Yaskawa INFORM job: A_ROOF_SIDE_0617_2_PAINT_59.JBI

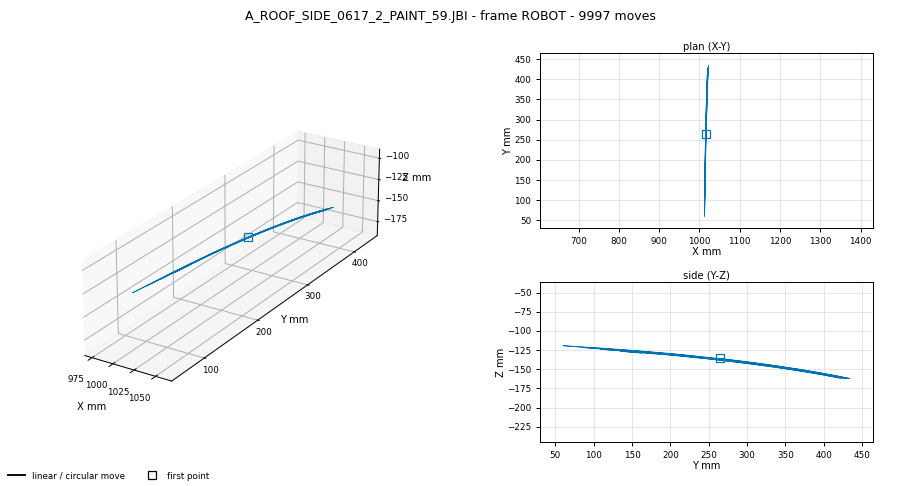
[picture p0: tool path of A_ROOF_SIDE_0617_2_PAINT_59.JBI in frame ROBOT, 9997 of 9997 moves have a stored position in this frame; points joined in program order, loops and branches not executed]
/JOB
//NAME A_ROOF_SIDE_0617_2_PAINT59
//POS
///NPOS 9997,0,0,0,0,0
///TOOL 1
///USER 0
///POSTYPE ROBOT
///RECTAN
///RCONF 1,0,0,0,0,0,0,0,0,0,0,0,0,0,0,0,0,0,0,0,0,0,0,0
C00000=1016.839,264.302,-135.724,169.198,51.675,159.894
C00001=1016.844,264.534,-135.751,169.203,51.669,159.893
C00002=1016.850,264.783,-135.779,169.208,51.663,159.893
C00003=1016.856,265.032,-135.809,169.212,51.657,159.892
C00004=1016.862,265.280,-135.837,169.217,51.651,159.892
C00005=1016.868,265.528,-135.866,169.222,51.644,159.891
C00006=1016.874,265.776,-135.895,169.228,51.638,159.891
C00007=1016.880,266.025,-135.923,169.233,51.632,159.891
C00008=1016.885,266.273,-135.953,169.237,51.626,159.890
C00009=1016.891,266.520,-135.982,169.242,51.620,159.890
C00010=1016.897,266.769,-136.010,169.247,51.614,159.889
C00011=1016.903,267.017,-136.039,169.252,51.607,159.889
C00012=1016.909,267.265,-136.068,169.257,51.602,159.888
C00013=1016.914,267.515,-136.097,169.262,51.596,159.888
C00014=1016.921,267.763,-136.126,169.267,51.589,159.887
C00015=1016.926,268.010,-136.155,169.272,51.583,159.887
C00016=1016.933,268.258,-136.184,169.277,51.577,159.887
C00017=1016.938,268.507,-136.213,169.282,51.571,159.886
C00018=1016.944,268.755,-136.242,169.287,51.565,159.886
C00019=1016.950,269.004,-136.271,169.292,51.559,159.885
C00020=1016.957,269.252,-136.300,169.297,51.553,159.885
C00021=1016.962,269.499,-136.329,169.302,51.547,159.884
C00022=1016.968,269.748,-136.358,169.306,51.541,159.884
C00023=1016.974,269.996,-136.387,169.311,51.535,159.883
C00024=1016.980,270.244,-136.417,169.317,51.529,159.883
C00025=1016.986,270.492,-136.446,169.322,51.523,159.883
C00026=1016.991,270.741,-136.476,169.327,51.517,159.882
C00027=1016.998,270.989,-136.505,169.332,51.511,159.882
C00028=1017.004,271.237,-136.534,169.337,51.505,159.882
C00029=1017.009,271.485,-136.563,169.342,51.500,159.881
C00030=1017.016,271.734,-136.592,169.347,51.494,159.881
C00031=1017.021,271.982,-136.622,169.352,51.488,159.880
C00032=1017.027,272.230,-136.651,169.357,51.482,159.880
C00033=1017.033,272.478,-136.680,169.362,51.476,159.880
C00034=1017.038,272.726,-136.709,169.367,51.470,159.879
C00035=1017.045,272.974,-136.738,169.372,51.464,159.879
C00036=1017.050,273.223,-136.768,169.377,51.459,159.879
C00037=1017.056,273.471,-136.797,169.382,51.453,159.878
C00038=1017.062,273.719,-136.827,169.387,51.447,159.878
C00039=1017.069,273.967,-136.856,169.392,51.441,159.877
C00040=1017.074,274.215,-136.886,169.398,51.435,159.877
C00041=1017.080,274.463,-136.915,169.403,51.429,159.877
C00042=1017.086,274.712,-136.945,169.408,51.423,159.876
C00043=1017.093,274.961,-136.974,169.414,51.418,159.876
C00044=1017.098,275.208,-137.005,169.419,51.412,159.876
C00045=1017.105,275.456,-137.034,169.424,51.407,159.875
C00046=1017.110,275.705,-137.063,169.429,51.401,159.875
C00047=1017.117,275.952,-137.093,169.434,51.395,159.875
C00048=1017.122,276.201,-137.123,169.439,51.389,159.874
C00049=1017.129,276.449,-137.152,169.444,51.384,159.874
C00050=1017.134,276.697,-137.182,169.449,51.378,159.874
C00051=1017.140,276.945,-137.212,169.454,51.372,159.873
C00052=1017.146,277.193,-137.241,169.459,51.367,159.873
C00053=1017.152,277.441,-137.271,169.464,51.361,159.873
C00054=1017.158,277.676,-137.300,169.469,51.357,159.872
C00055=1017.163,277.911,-137.328,169.474,51.351,159.872
C00056=1017.168,278.147,-137.356,169.479,51.346,159.872
C00057=1017.175,278.382,-137.385,169.484,51.341,159.871
C00058=1017.180,278.617,-137.413,169.489,51.335,159.871
C00059=1017.186,278.852,-137.442,169.494,51.330,159.871
C00060=1017.191,279.088,-137.470,169.498,51.325,159.871
C00061=1017.197,279.322,-137.498,169.503,51.319,159.870
C00062=1017.203,279.571,-137.528,169.509,51.314,159.870
C00063=1017.209,279.819,-137.558,169.514,51.308,159.870
C00064=1017.215,280.067,-137.588,169.519,51.303,159.869
C00065=1017.221,280.315,-137.618,169.524,51.297,159.869
C00066=1017.227,280.563,-137.648,169.530,51.292,159.869
C00067=1017.233,280.811,-137.678,169.535,51.286,159.868
C00068=1017.239,281.060,-137.708,169.540,51.281,159.868
C00069=1017.245,281.307,-137.738,169.546,51.276,159.868
C00070=1017.252,281.555,-137.768,169.551,51.270,159.868
C00071=1017.257,281.803,-137.798,169.556,51.265,159.868
C00072=1017.264,282.052,-137.829,169.561,51.259,159.867
C00073=1017.269,282.300,-137.859,169.566,51.254,159.867
C00074=1017.276,282.547,-137.889,169.572,51.249,159.867
C00075=1017.282,282.796,-137.919,169.577,51.243,159.866
C00076=1017.288,283.044,-137.949,169.582,51.238,159.866
C00077=1017.294,283.292,-137.979,169.588,51.233,159.866
C00078=1017.300,283.540,-138.009,169.593,51.227,159.866
C00079=1017.307,283.788,-138.040,169.598,51.222,159.865
C00080=1017.312,284.036,-138.070,169.604,51.217,159.865
C00081=1017.319,284.285,-138.100,169.609,51.211,159.865
C00082=1017.325,284.533,-138.130,169.614,51.206,159.865
C00083=1017.331,284.780,-138.160,169.619,51.201,159.864
C00084=1017.337,285.028,-138.191,169.625,51.196,159.864
C00085=1017.343,285.277,-138.221,169.629,51.191,159.864
C00086=1017.349,285.525,-138.252,169.634,51.185,159.864
C00087=1017.355,285.773,-138.282,169.640,51.180,159.863
C00088=1017.362,286.020,-138.313,169.645,51.175,159.863
C00089=1017.367,286.268,-138.344,169.651,51.170,159.863
C00090=1017.374,286.517,-138.375,169.656,51.165,159.863
C00091=1017.380,286.764,-138.405,169.661,51.160,159.863
C00092=1017.386,287.013,-138.436,169.667,51.155,159.862
C00093=1017.392,287.261,-138.466,169.672,51.149,159.862
C00094=1017.398,287.509,-138.496,169.678,51.144,159.862
C00095=1017.404,287.757,-138.527,169.683,51.139,159.862
C00096=1017.410,288.004,-138.558,169.689,51.134,159.862
C00097=1017.417,288.253,-138.589,169.694,51.129,159.861
C00098=1017.422,288.501,-138.619,169.699,51.124,159.861
C00099=1017.429,288.749,-138.650,169.705,51.119,159.861
C00100=1017.434,288.997,-138.682,169.710,51.114,159.861
C00101=1017.441,289.245,-138.712,169.716,51.108,159.861
C00102=1017.446,289.493,-138.743,169.721,51.103,159.861
C00103=1017.453,289.741,-138.774,169.726,51.099,159.860
C00104=1017.459,289.989,-138.804,169.731,51.094,159.860
C00105=1017.465,290.237,-138.835,169.737,51.089,159.860
C00106=1017.472,290.485,-138.866,169.742,51.084,159.860
C00107=1017.478,290.733,-138.897,169.748,51.079,159.860
C00108=1017.484,290.980,-138.928,169.753,51.074,159.860
C00109=1017.490,291.229,-138.959,169.759,51.069,159.859
C00110=1017.496,291.477,-138.989,169.764,51.064,159.859
C00111=1017.502,291.725,-139.021,169.770,51.059,159.859
C00112=1017.508,291.972,-139.052,169.775,51.054,159.859
C00113=1017.515,292.221,-139.083,169.781,51.049,159.859
C00114=1017.520,292.462,-139.113,169.786,51.045,159.859
C00115=1017.527,292.703,-139.143,169.791,51.040,159.858
C00116=1017.533,292.944,-139.173,169.797,51.035,159.859
C00117=1017.539,293.186,-139.204,169.802,51.030,159.858
C00118=1017.545,293.427,-139.235,169.807,51.026,159.858
C00119=1017.551,293.668,-139.265,169.812,51.021,159.858
C00120=1017.556,293.910,-139.295,169.818,51.017,159.858
C00121=1017.563,294.151,-139.327,169.823,51.012,159.858
C00122=1017.568,294.398,-139.358,169.829,51.007,159.858
C00123=1017.574,294.647,-139.390,169.834,51.003,159.858
C00124=1017.580,294.894,-139.421,169.840,50.998,159.858
C00125=1017.586,295.143,-139.453,169.846,50.993,159.858
C00126=1017.593,295.390,-139.484,169.851,50.988,159.857
C00127=1017.598,295.638,-139.516,169.856,50.984,159.857
C00128=1017.605,295.886,-139.547,169.861,50.979,159.857
C00129=1017.611,296.134,-139.579,169.867,50.975,159.857
C00130=1017.617,296.381,-139.610,169.873,50.970,159.857
C00131=1017.623,296.629,-139.642,169.879,50.965,159.857
C00132=1017.630,296.877,-139.674,169.884,50.961,159.857
C00133=1017.635,297.125,-139.705,169.890,50.956,159.857
C00134=1017.641,297.373,-139.737,169.896,50.951,159.857
C00135=1017.648,297.621,-139.769,169.900,50.947,159.857
C00136=1017.654,297.869,-139.801,169.906,50.943,159.857
C00137=1017.660,298.116,-139.832,169.912,50.938,159.857
C00138=1017.666,298.365,-139.864,169.918,50.933,159.857
C00139=1017.673,298.613,-139.895,169.923,50.929,159.857
C00140=1017.679,298.861,-139.927,169.929,50.924,159.857
C00141=1017.685,299.109,-139.959,169.935,50.920,159.857
C00142=1017.691,299.356,-139.991,169.941,50.915,159.856
C00143=1017.697,299.604,-140.022,169.945,50.911,159.856
C00144=1017.703,299.852,-140.054,169.951,50.906,159.856
C00145=1017.710,300.100,-140.087,169.957,50.902,159.856
C00146=1017.716,300.348,-140.118,169.963,50.898,159.856
C00147=1017.722,300.596,-140.150,169.969,50.893,159.856
C00148=1017.729,300.843,-140.181,169.974,50.888,159.856
C00149=1017.734,301.091,-140.213,169.980,50.884,159.856
C00150=1017.742,301.339,-140.245,169.986,50.879,159.856
C00151=1017.748,301.587,-140.278,169.992,50.875,159.856
C00152=1017.754,301.835,-140.309,169.997,50.871,159.856
C00153=1017.761,302.082,-140.342,170.002,50.866,159.856
C00154=1017.767,302.331,-140.374,170.008,50.862,159.856
C00155=1017.773,302.579,-140.405,170.014,50.857,159.856
C00156=1017.780,302.826,-140.438,170.020,50.853,159.856
C00157=1017.786,303.074,-140.469,170.026,50.849,159.856
C00158=1017.792,303.322,-140.501,170.032,50.844,159.856
C00159=1017.799,303.570,-140.533,170.037,50.840,159.856
C00160=1017.805,303.818,-140.566,170.043,50.835,159.856
C00161=1017.812,304.065,-140.598,170.049,50.831,159.856
C00162=1017.818,304.313,-140.630,170.055,50.827,159.856
C00163=1017.825,304.561,-140.662,170.060,50.822,159.856
C00164=1017.831,304.809,-140.694,170.066,50.818,159.856
C00165=1017.837,305.057,-140.726,170.072,50.814,159.856
C00166=1017.844,305.304,-140.758,170.078,50.810,159.856
C00167=1017.851,305.552,-140.791,170.084,50.805,159.856
C00168=1017.857,305.800,-140.823,170.089,50.801,159.856
C00169=1017.864,306.047,-140.855,170.095,50.797,159.856
C00170=1017.870,306.296,-140.887,170.101,50.792,159.856
C00171=1017.877,306.543,-140.919,170.107,50.789,159.857
C00172=1017.883,306.791,-140.951,170.113,50.784,159.857
C00173=1017.890,307.038,-140.983,170.119,50.780,159.857
C00174=1017.896,307.291,-141.017,170.125,50.775,159.857
C00175=1017.903,307.544,-141.049,170.131,50.771,159.857
C00176=1017.910,307.796,-141.083,170.137,50.767,159.857
C00177=1017.917,308.049,-141.116,170.143,50.763,159.857
C00178=1017.923,308.297,-141.147,170.149,50.758,159.857
C00179=1017.930,308.544,-141.180,170.155,50.754,159.857
C00180=1017.937,308.792,-141.212,170.161,50.750,159.857
C00181=1017.943,309.039,-141.245,170.167,50.746,159.857
C00182=1017.950,309.287,-141.278,170.172,50.741,159.857
C00183=1017.957,309.535,-141.309,170.179,50.738,159.857
C00184=1017.963,309.783,-141.342,170.185,50.733,159.857
C00185=1017.969,310.031,-141.375,170.190,50.730,159.857
C00186=1017.976,310.278,-141.408,170.196,50.726,159.858
C00187=1017.981,310.525,-141.442,170.202,50.722,159.858
C00188=1017.988,310.774,-141.475,170.208,50.718,159.858
C00189=1017.994,311.021,-141.508,170.214,50.714,159.858
C00190=1018.001,311.269,-141.540,170.220,50.710,159.858
C00191=1018.007,311.517,-141.573,170.225,50.706,159.858
C00192=1018.013,311.764,-141.607,170.232,50.703,159.858
C00193=1018.020,312.012,-141.640,170.238,50.698,159.858
C00194=1018.026,312.260,-141.673,170.244,50.695,159.859
C00195=1018.033,312.507,-141.706,170.250,50.691,159.859
C00196=1018.039,312.754,-141.739,170.256,50.687,159.859
C00197=1018.045,313.003,-141.773,170.262,50.683,159.859
C00198=1018.051,313.250,-141.806,170.267,50.679,159.859
C00199=1018.058,313.497,-141.839,170.274,50.676,159.859
C00200=1018.065,313.746,-141.872,170.280,50.672,159.859
C00201=1018.072,313.993,-141.906,170.286,50.668,159.860
C00202=1018.077,314.241,-141.939,170.292,50.664,159.860
C00203=1018.084,314.489,-141.972,170.298,50.660,159.860
C00204=1018.091,314.736,-142.006,170.304,50.656,159.860
C00205=1018.097,314.983,-142.038,170.311,50.652,159.860
C00206=1018.103,315.231,-142.073,170.316,50.649,159.860
C00207=1018.110,315.479,-142.105,170.322,50.645,159.861
C00208=1018.117,315.727,-142.139,170.328,50.642,159.861
C00209=1018.123,315.974,-142.172,170.335,50.638,159.861
C00210=1018.130,316.221,-142.205,170.341,50.634,159.861
C00211=1018.136,316.470,-142.239,170.347,50.630,159.861
C00212=1018.143,316.717,-142.273,170.353,50.627,159.862
C00213=1018.149,316.965,-142.306,170.360,50.623,159.862
C00214=1018.156,317.212,-142.339,170.366,50.619,159.862
C00215=1018.162,317.460,-142.374,170.372,50.615,159.862
C00216=1018.169,317.708,-142.406,170.377,50.612,159.862
C00217=1018.176,317.955,-142.440,170.384,50.608,159.863
C00218=1018.183,318.202,-142.474,170.390,50.605,159.863
C00219=1018.189,318.451,-142.507,170.396,50.601,159.863
C00220=1018.196,318.699,-142.541,170.403,50.598,159.863
C00221=1018.203,318.946,-142.575,170.409,50.594,159.864
C00222=1018.209,319.194,-142.608,170.415,50.590,159.864
C00223=1018.216,319.441,-142.641,170.421,50.587,159.864
C00224=1018.222,319.689,-142.676,170.428,50.583,159.864
C00225=1018.230,319.937,-142.709,170.434,50.579,159.864
C00226=1018.236,320.184,-142.742,170.441,50.576,159.865
C00227=1018.243,320.432,-142.776,170.447,50.572,159.865
C00228=1018.249,320.679,-142.810,170.453,50.569,159.865
C00229=1018.256,320.927,-142.844,170.459,50.565,159.865
C00230=1018.263,321.174,-142.878,170.466,50.562,159.866
C00231=1018.271,321.422,-142.912,170.472,50.558,159.866
C00232=1018.276,321.669,-142.946,170.478,50.554,159.866
C00233=1018.284,321.917,-142.979,170.484,50.552,159.867
C00234=1018.291,322.175,-143.014,170.491,50.548,159.867
C00235=1018.298,322.433,-143.049,170.498,50.544,159.867
C00236=1018.305,322.691,-143.084,170.504,50.540,159.867
C00237=1018.312,322.949,-143.120,170.511,50.537,159.868
C00238=1018.319,323.197,-143.154,170.518,50.533,159.868
C00239=1018.326,323.444,-143.188,170.523,50.530,159.868
C00240=1018.333,323.691,-143.222,170.530,50.527,159.868
C00241=1018.340,323.939,-143.255,170.536,50.523,159.869
C00242=1018.346,324.187,-143.290,170.542,50.520,159.869
C00243=1018.354,324.435,-143.324,170.549,50.516,159.869
C00244=1018.361,324.682,-143.358,170.555,50.513,159.870
C00245=1018.368,324.929,-143.392,170.562,50.509,159.870
C00246=1018.375,325.177,-143.426,170.568,50.506,159.870
C00247=1018.381,325.424,-143.460,170.576,50.503,159.871
C00248=1018.389,325.672,-143.494,170.582,50.499,159.871
C00249=1018.395,325.920,-143.528,170.589,50.496,159.871
C00250=1018.403,326.167,-143.563,170.595,50.492,159.871
C00251=1018.410,326.415,-143.597,170.602,50.489,159.872
C00252=1018.416,326.662,-143.632,170.608,50.486,159.872
C00253=1018.423,326.910,-143.666,170.614,50.483,159.873
C00254=1018.430,327.157,-143.701,170.620,50.480,159.873
C00255=1018.437,327.405,-143.735,170.627,50.477,159.873
C00256=1018.444,327.652,-143.770,170.633,50.473,159.874
C00257=1018.451,327.900,-143.804,170.640,50.470,159.874
C00258=1018.458,328.148,-143.839,170.647,50.467,159.874
C00259=1018.464,328.395,-143.874,170.653,50.464,159.875
C00260=1018.471,328.642,-143.908,170.659,50.461,159.875
C00261=1018.478,328.889,-143.943,170.666,50.457,159.875
C00262=1018.484,329.137,-143.977,170.673,50.454,159.876
C00263=1018.492,329.385,-144.013,170.679,50.451,159.876
C00264=1018.499,329.632,-144.047,170.686,50.448,159.877
C00265=1018.506,329.880,-144.082,170.693,50.445,159.877
C00266=1018.512,330.128,-144.117,170.699,50.442,159.877
C00267=1018.520,330.375,-144.151,170.706,50.439,159.878
C00268=1018.527,330.622,-144.187,170.713,50.436,159.878
C00269=1018.533,330.869,-144.222,170.719,50.433,159.879
C00270=1018.540,331.117,-144.256,170.726,50.430,159.879
C00271=1018.547,331.364,-144.291,170.732,50.427,159.879
C00272=1018.554,331.612,-144.326,170.739,50.424,159.880
C00273=1018.561,331.859,-144.361,170.746,50.421,159.880
C00274=1018.569,332.107,-144.396,170.753,50.418,159.881
C00275=1018.576,332.354,-144.431,170.759,50.415,159.881
C00276=1018.583,332.602,-144.466,170.766,50.412,159.882
C00277=1018.589,332.849,-144.501,170.773,50.409,159.882
C00278=1018.596,333.096,-144.536,170.780,50.407,159.883
C00279=1018.603,333.344,-144.571,170.786,50.403,159.883
C00280=1018.610,333.592,-144.607,170.793,50.400,159.883
C00281=1018.617,333.839,-144.642,170.800,50.397,159.884
C00282=1018.625,334.086,-144.677,170.807,50.395,159.884
C00283=1018.631,334.334,-144.712,170.813,50.392,159.885
C00284=1018.639,334.581,-144.748,170.820,50.389,159.885
C00285=1018.646,334.828,-144.783,170.827,50.386,159.886
C00286=1018.652,335.076,-144.818,170.833,50.383,159.886
C00287=1018.659,335.323,-144.853,170.841,50.381,159.887
C00288=1018.667,335.571,-144.890,170.848,50.377,159.887
C00289=1018.674,335.818,-144.925,170.855,50.375,159.888
C00290=1018.680,336.065,-144.960,170.862,50.372,159.888
C00291=1018.688,336.313,-144.996,170.869,50.370,159.889
C00292=1018.695,336.560,-145.031,170.875,50.366,159.889
C00293=1018.702,336.808,-145.066,170.882,50.364,159.890
C00294=1018.709,337.061,-145.104,170.889,50.361,159.890
C00295=1018.717,337.315,-145.140,170.896,50.359,159.891
C00296=1018.724,337.568,-145.176,170.904,50.355,159.891
C00297=1018.731,337.823,-145.213,170.911,50.353,159.892
C00298=1018.738,338.069,-145.249,170.917,50.350,159.892
C00299=1018.745,338.317,-145.284,170.924,50.347,159.893
C00300=1018.753,338.564,-145.320,170.931,50.345,159.894
C00301=1018.760,338.811,-145.355,170.938,50.342,159.894
C00302=1018.767,339.059,-145.392,170.945,50.339,159.895
C00303=1018.774,339.306,-145.427,170.952,50.337,159.895
C00304=1018.782,339.554,-145.463,170.959,50.334,159.896
C00305=1018.789,339.801,-145.499,170.967,50.331,159.896
C00306=1018.796,340.048,-145.535,170.974,50.329,159.897
C00307=1018.802,340.296,-145.571,170.981,50.326,159.897
C00308=1018.810,340.543,-145.607,170.988,50.324,159.898
C00309=1018.817,340.790,-145.643,170.995,50.321,159.899
C00310=1018.825,341.037,-145.679,171.002,50.319,159.899
C00311=1018.832,341.284,-145.715,171.009,50.317,159.900
C00312=1018.839,341.532,-145.752,171.016,50.314,159.900
C00313=1018.846,341.779,-145.788,171.023,50.312,159.901
C00314=1018.854,342.026,-145.824,171.029,50.309,159.901
C00315=1018.861,342.274,-145.859,171.038,50.306,159.902
C00316=1018.867,342.521,-145.896,171.045,50.303,159.903
C00317=1018.875,342.769,-145.932,171.052,50.302,159.904
C00318=1018.883,343.015,-145.969,171.059,50.299,159.904
C00319=1018.889,343.262,-146.005,171.066,50.297,159.905
C00320=1018.897,343.510,-146.042,171.073,50.294,159.905
C00321=1018.905,343.757,-146.078,171.080,50.292,159.906
C00322=1018.912,344.004,-146.114,171.088,50.289,159.907
C00323=1018.919,344.252,-146.150,171.095,50.287,159.907
C00324=1018.926,344.499,-146.187,171.102,50.284,159.908
C00325=1018.934,344.747,-146.223,171.109,50.283,159.909
C00326=1018.941,344.993,-146.260,171.116,50.280,159.909
C00327=1018.948,345.241,-146.296,171.123,50.278,159.910
C00328=1018.956,345.488,-146.332,171.131,50.275,159.911
C00329=1018.963,345.736,-146.369,171.139,50.272,159.911
C00330=1018.971,345.983,-146.406,171.146,50.271,159.912
C00331=1018.978,346.229,-146.442,171.153,50.268,159.913
C00332=1018.985,346.477,-146.479,171.160,50.266,159.913
C00333=1018.993,346.724,-146.516,171.168,50.264,159.914
C00334=1019.001,346.971,-146.552,171.175,50.261,159.915
C00335=1019.008,347.219,-146.590,171.183,50.259,159.915
C00336=1019.015,347.466,-146.626,171.190,50.257,159.916
C00337=1019.023,347.713,-146.663,171.197,50.255,159.917
C00338=1019.030,347.960,-146.699,171.204,50.253,159.917
C00339=1019.037,348.207,-146.737,171.212,50.250,159.918
C00340=1019.045,348.454,-146.774,171.220,50.248,159.919
C00341=1019.052,348.702,-146.810,171.227,50.246,159.920
C00342=1019.059,348.949,-146.848,171.234,50.244,159.920
C00343=1019.067,349.196,-146.885,171.242,50.242,159.921
C00344=1019.074,349.443,-146.922,171.249,50.239,159.922
C00345=1019.082,349.690,-146.959,171.257,50.238,159.923
C00346=1019.089,349.937,-146.996,171.264,50.236,159.923
C00347=1019.097,350.184,-147.034,171.272,50.233,159.924
C00348=1019.105,350.431,-147.071,171.280,50.231,159.925
C00349=1019.111,350.679,-147.107,171.287,50.230,159.926
C00350=1019.119,350.926,-147.144,171.294,50.227,159.926
C00351=1019.127,351.173,-147.182,171.302,50.225,159.927
C00352=1019.134,351.420,-147.219,171.310,50.223,159.928
C00353=1019.142,351.667,-147.256,171.317,50.221,159.929
C00354=1019.150,351.918,-147.294,171.326,50.219,159.930
C00355=1019.157,352.169,-147.332,171.333,50.217,159.930
C00356=1019.165,352.419,-147.370,171.340,50.215,159.931
C00357=1019.173,352.671,-147.408,171.348,50.213,159.932
C00358=1019.181,352.918,-147.445,171.356,50.211,159.933
C00359=1019.189,353.165,-147.482,171.363,50.209,159.933
C00360=1019.196,353.411,-147.521,171.372,50.207,159.934
C00361=1019.203,353.659,-147.558,171.379,50.205,159.935
C00362=1019.212,353.906,-147.595,171.386,50.204,159.936
C00363=1019.219,354.153,-147.633,171.395,50.201,159.937
C00364=1019.226,354.400,-147.670,171.402,50.200,159.938
C00365=1019.234,354.647,-147.709,171.410,50.198,159.938
C00366=1019.242,354.894,-147.746,171.418,50.196,159.939
C00367=1019.250,355.142,-147.784,171.425,50.194,159.940
C00368=1019.257,355.388,-147.822,171.433,50.193,159.941
C00369=1019.265,355.635,-147.859,171.442,50.191,159.942
C00370=1019.273,355.882,-147.898,171.449,50.189,159.943
C00371=1019.281,356.129,-147.935,171.456,50.187,159.944
C00372=1019.288,356.376,-147.972,171.465,50.185,159.944
C00373=1019.296,356.624,-148.011,171.473,50.184,159.945
C00374=1019.304,356.870,-148.049,171.481,50.182,159.946
C00375=1019.311,357.117,-148.087,171.488,50.180,159.947
C00376=1019.320,357.364,-148.125,171.496,50.178,159.948
C00377=1019.327,357.611,-148.162,171.504,50.176,159.949
C00378=1019.335,357.858,-148.200,171.512,50.175,159.950
C00379=1019.343,358.105,-148.239,171.521,50.173,159.951
C00380=1019.350,358.352,-148.277,171.528,50.171,159.952
C00381=1019.358,358.599,-148.315,171.535,50.169,159.953
C00382=1019.366,358.846,-148.353,171.544,50.168,159.954
C00383=1019.374,359.093,-148.391,171.552,50.166,159.954
C00384=1019.382,359.340,-148.429,171.560,50.165,159.955
C00385=1019.390,359.587,-148.468,171.568,50.163,159.956
C00386=1019.397,359.834,-148.506,171.577,50.161,159.957
C00387=1019.406,360.081,-148.544,171.584,50.160,159.958
C00388=1019.413,360.327,-148.583,171.593,50.158,159.959
C00389=1019.421,360.575,-148.622,171.600,50.157,159.960
C00390=1019.428,360.821,-148.660,171.608,50.156,159.961
C00391=1019.436,361.069,-148.699,171.617,50.153,159.962
C00392=1019.444,361.315,-148.737,171.624,50.152,159.963
C00393=1019.452,361.562,-148.776,171.633,50.151,159.964
C00394=1019.460,361.809,-148.815,171.641,50.150,159.965
C00395=1019.468,362.056,-148.853,171.649,50.147,159.966
C00396=1019.476,362.303,-148.892,171.657,50.146,159.967
C00397=1019.484,362.550,-148.930,171.666,50.145,159.968
C00398=1019.491,362.797,-148.969,171.674,50.144,159.969
C00399=1019.500,363.043,-149.009,171.682,50.142,159.970
C00400=1019.508,363.291,-149.047,171.690,50.141,159.971
C00401=1019.515,363.537,-149.085,171.699,50.139,159.972
C00402=1019.524,363.784,-149.125,171.707,50.138,159.973
C00403=1019.532,364.031,-149.163,171.716,50.137,159.974
C00404=1019.540,364.277,-149.202,171.724,50.135,159.976
C00405=1019.548,364.524,-149.241,171.732,50.134,159.977
C00406=1019.555,364.772,-149.280,171.741,50.132,159.978
C00407=1019.564,365.018,-149.319,171.749,50.131,159.979
C00408=1019.572,365.265,-149.358,171.757,50.130,159.980
C00409=1019.580,365.512,-149.397,171.765,50.128,159.981
C00410=1019.588,365.758,-149.436,171.774,50.127,159.982
C00411=1019.596,366.005,-149.475,171.783,50.125,159.983
C00412=1019.605,366.252,-149.514,171.790,50.124,159.984
C00413=1019.613,366.499,-149.553,171.800,50.123,159.985
C00414=1019.621,366.757,-149.594,171.808,50.122,159.986
C00415=1019.630,367.016,-149.636,171.817,50.120,159.987
C00416=1019.639,367.274,-149.676,171.826,50.119,159.989
C00417=1019.647,367.532,-149.718,171.835,50.118,159.990
C00418=1019.655,367.779,-149.757,171.844,50.116,159.991
C00419=1019.664,368.025,-149.796,171.852,50.116,159.992
C00420=1019.672,368.272,-149.836,171.861,50.114,159.993
C00421=1019.680,368.519,-149.875,171.870,50.113,159.994
C00422=1019.688,368.766,-149.915,171.878,50.112,159.995
C00423=1019.696,369.012,-149.955,171.887,50.111,159.997
C00424=1019.704,369.259,-149.995,171.896,50.110,159.998
C00425=1019.712,369.506,-150.034,171.904,50.109,159.999
C00426=1019.721,369.752,-150.073,171.913,50.107,160.000
C00427=1019.729,369.999,-150.113,171.922,50.107,160.001
C00428=1019.737,370.245,-150.153,171.930,50.106,160.003
C00429=1019.745,370.492,-150.193,171.939,50.104,160.004
C00430=1019.754,370.739,-150.233,171.948,50.103,160.005
C00431=1019.762,370.986,-150.273,171.957,50.103,160.006
C00432=1019.771,371.232,-150.313,171.965,50.101,160.007
C00433=1019.778,371.479,-150.353,171.974,50.100,160.009
C00434=1019.787,371.726,-150.392,171.983,50.100,160.010
C00435=1019.795,371.972,-150.433,171.992,50.099,160.011
C00436=1019.804,372.219,-150.472,172.000,50.098,160.012
C00437=1019.813,372.465,-150.512,172.009,50.096,160.013
C00438=1019.820,372.712,-150.552,172.018,50.096,160.015
C00439=1019.829,372.958,-150.592,172.027,50.095,160.016
C00440=1019.837,373.206,-150.633,172.037,50.094,160.017
C00441=1019.846,373.452,-150.673,172.046,50.093,160.019
C00442=1019.854,373.699,-150.713,172.054,50.092,160.020
C00443=1019.863,373.945,-150.753,172.063,50.091,160.021
C00444=1019.871,374.192,-150.793,172.072,50.090,160.022
C00445=1019.880,374.438,-150.833,172.081,50.089,160.024
C00446=1019.888,374.685,-150.874,172.090,50.088,160.025
C00447=1019.897,374.931,-150.914,172.100,50.087,160.026
C00448=1019.905,375.179,-150.954,172.109,50.087,160.027
C00449=1019.914,375.425,-150.994,172.118,50.086,160.029
C00450=1019.923,375.671,-151.034,172.126,50.086,160.030
C00451=1019.932,375.918,-151.075,172.136,50.085,160.031
C00452=1019.940,376.164,-151.116,172.145,50.084,160.033
C00453=1019.949,376.411,-151.156,172.154,50.083,160.034
C00454=1019.957,376.657,-151.197,172.163,50.082,160.036
C00455=1019.966,376.904,-151.238,172.173,50.082,160.037
C00456=1019.974,377.150,-151.279,172.182,50.081,160.038
C00457=1019.982,377.397,-151.320,172.191,50.080,160.040
C00458=1019.991,377.643,-151.360,172.201,50.080,160.041
C00459=1020.000,377.889,-151.401,172.210,50.079,160.042
C00460=1020.008,378.136,-151.442,172.219,50.079,160.044
C00461=1020.017,378.383,-151.483,172.229,50.078,160.045
C00462=1020.025,378.630,-151.524,172.238,50.077,160.047
C00463=1020.034,378.875,-151.565,172.247,50.076,160.048
C00464=1020.043,379.122,-151.606,172.257,50.076,160.049
C00465=1020.052,379.369,-151.647,172.266,50.075,160.051
C00466=1020.060,379.615,-151.688,172.275,50.075,160.052
C00467=1020.069,379.862,-151.729,172.285,50.074,160.054
C00468=1020.078,380.108,-151.770,172.295,50.074,160.055
C00469=1020.086,380.354,-151.811,172.304,50.073,160.057
C00470=1020.095,380.600,-151.853,172.313,50.073,160.058
C00471=1020.104,380.847,-151.894,172.323,50.072,160.060
C00472=1020.113,381.094,-151.935,172.332,50.072,160.061
C00473=1020.122,381.339,-151.976,172.342,50.072,160.063
C00474=1020.132,381.620,-152.023,172.353,50.071,160.064
C00475=1020.141,381.901,-152.070,172.364,50.070,160.066
C00476=1020.152,382.181,-152.118,172.375,50.070,160.068
C00477=1020.162,382.461,-152.165,172.385,50.069,160.069
C00478=1020.171,382.708,-152.206,172.396,50.069,160.071
C00479=1020.181,382.954,-152.248,172.405,50.068,160.072
C00480=1020.189,383.201,-152.289,172.415,50.068,160.074
C00481=1020.198,383.447,-152.330,172.425,50.068,160.075
C00482=1020.207,383.694,-152.372,172.434,50.068,160.077
C00483=1020.216,383.940,-152.414,172.445,50.067,160.079
C00484=1020.226,384.186,-152.455,172.454,50.067,160.080
C00485=1020.235,384.432,-152.497,172.464,50.066,160.082
C00486=1020.243,384.679,-152.538,172.473,50.066,160.083
C00487=1020.252,384.925,-152.580,172.484,50.066,160.085
C00488=1020.261,385.171,-152.622,172.494,50.065,160.086
C00489=1020.272,385.418,-152.663,172.503,50.065,160.088
C00490=1020.280,385.664,-152.706,172.514,50.065,160.090
C00491=1020.289,385.911,-152.748,172.524,50.065,160.091
C00492=1020.298,386.157,-152.790,172.533,50.064,160.093
C00493=1020.307,386.403,-152.832,172.543,50.065,160.094
C00494=1020.316,386.649,-152.874,172.554,50.064,160.096
C00495=1020.325,386.895,-152.916,172.564,50.064,160.098
C00496=1020.334,387.141,-152.958,172.573,50.064,160.099
C00497=1020.344,387.388,-153.001,172.584,50.064,160.101
C00498=1020.353,387.634,-153.042,172.594,50.064,160.103
C00499=1020.362,387.880,-153.085,172.604,50.063,160.104
C00500=1020.371,388.126,-153.127,172.614,50.063,160.106
C00501=1020.381,388.373,-153.169,172.624,50.064,160.108
C00502=1020.390,388.618,-153.212,172.635,50.063,160.109
C00503=1020.399,388.864,-153.255,172.645,50.063,160.111
C00504=1020.408,389.111,-153.297,172.656,50.063,160.113
C00505=1020.418,389.357,-153.339,172.666,50.063,160.114
C00506=1020.427,389.603,-153.382,172.676,50.063,160.116
C00507=1020.436,389.849,-153.424,172.686,50.063,160.118
C00508=1020.445,390.095,-153.468,172.696,50.063,160.120
C00509=1020.454,390.341,-153.510,172.707,50.063,160.121
C00510=1020.464,390.588,-153.553,172.717,50.064,160.123
C00511=1020.474,390.833,-153.595,172.728,50.063,160.125
C00512=1020.483,391.080,-153.639,172.739,50.063,160.127
C00513=1020.492,391.326,-153.681,172.749,50.063,160.128
C00514=1020.502,391.572,-153.724,172.760,50.063,160.130
C00515=1020.511,391.817,-153.767,172.770,50.064,160.132
C00516=1020.521,392.064,-153.810,172.781,50.063,160.134
C00517=1020.530,392.310,-153.853,172.791,50.064,160.136
C00518=1020.539,392.556,-153.896,172.802,50.064,160.137
C00519=1020.549,392.802,-153.939,172.813,50.064,160.139
C00520=1020.558,393.048,-153.982,172.823,50.065,160.141
C00521=1020.568,393.295,-154.025,172.834,50.065,160.143
C00522=1020.577,393.540,-154.069,172.844,50.065,160.145
C00523=1020.587,393.786,-154.112,172.855,50.065,160.147
C00524=1020.597,394.032,-154.155,172.866,50.065,160.148
C00525=1020.606,394.278,-154.199,172.876,50.066,160.150
C00526=1020.615,394.524,-154.242,172.887,50.066,160.152
C00527=1020.626,394.770,-154.285,172.898,50.066,160.154
C00528=1020.634,395.016,-154.329,172.910,50.067,160.156
C00529=1020.644,395.262,-154.372,172.920,50.067,160.158
C00530=1020.654,395.508,-154.416,172.931,50.067,160.160
C00531=1020.664,395.754,-154.459,172.942,50.068,160.162
C00532=1020.674,396.000,-154.503,172.953,50.068,160.164
C00533=1020.683,396.246,-154.547,172.963,50.068,160.165
C00534=1020.699,396.634,-154.616,172.981,50.069,160.169
C00535=1020.714,397.023,-154.685,172.998,50.069,160.172
C00536=1020.730,397.413,-154.754,173.016,50.070,160.175
C00537=1020.745,397.801,-154.823,173.033,50.071,160.178
C00538=1020.754,398.047,-154.868,173.045,50.071,160.180
C00539=1020.764,398.293,-154.911,173.056,50.072,160.182
C00540=1020.774,398.540,-154.956,173.067,50.072,160.184
C00541=1020.784,398.786,-154.999,173.079,50.073,160.186
C00542=1020.794,399.031,-155.044,173.090,50.073,160.188
C00543=1020.804,399.277,-155.087,173.102,50.074,160.190
C00544=1020.814,399.522,-155.132,173.113,50.074,160.192
C00545=1020.823,399.769,-155.176,173.125,50.075,160.194
C00546=1020.834,400.014,-155.221,173.136,50.076,160.196
C00547=1020.843,400.260,-155.265,173.147,50.076,160.198
C00548=1020.853,400.505,-155.310,173.159,50.077,160.201
C00549=1020.864,400.752,-155.353,173.170,50.077,160.203
C00550=1020.874,400.997,-155.398,173.181,50.078,160.205
C00551=1020.883,401.243,-155.443,173.193,50.079,160.207
C00552=1020.893,401.488,-155.488,173.205,50.080,160.209
C00553=1020.903,401.734,-155.532,173.216,50.080,160.211
C00554=1020.914,401.980,-155.577,173.228,50.081,160.213
C00555=1020.923,402.225,-155.622,173.239,50.082,160.215
C00556=1020.933,402.471,-155.666,173.251,50.083,160.217
C00557=1020.943,402.718,-155.711,173.263,50.083,160.220
C00558=1020.954,402.962,-155.756,173.275,50.084,160.222
C00559=1020.964,403.208,-155.801,173.286,50.085,160.224
C00560=1020.974,403.454,-155.846,173.298,50.086,160.226
C00561=1020.984,403.700,-155.891,173.310,50.087,160.228
C00562=1020.994,403.946,-155.936,173.322,50.087,160.231
C00563=1021.004,404.191,-155.981,173.334,50.088,160.233
C00564=1021.015,404.437,-156.027,173.346,50.089,160.235
C00565=1021.025,404.682,-156.071,173.357,50.090,160.237
C00566=1021.033,404.893,-156.110,173.368,50.091,160.239
C00567=1021.042,405.102,-156.149,173.378,50.092,160.241
C00568=1021.051,405.313,-156.187,173.388,50.092,160.243
C00569=1021.060,405.522,-156.226,173.398,50.093,160.245
C00570=1021.069,405.732,-156.265,173.409,50.094,160.247
C00571=1021.078,405.943,-156.303,173.419,50.095,160.249
C00572=1021.086,406.153,-156.342,173.430,50.096,160.251
C00573=1021.097,406.363,-156.381,173.440,50.096,160.253
C00574=1021.106,406.608,-156.426,173.453,50.097,160.255
C00575=1021.117,406.854,-156.472,173.465,50.099,160.258
C00576=1021.128,407.100,-156.518,173.477,50.099,160.260
C00577=1021.138,407.346,-156.563,173.489,50.100,160.262
C00578=1021.148,407.591,-156.609,173.502,50.101,160.265
C00579=1021.159,407.836,-156.654,173.514,50.102,160.267
C00580=1021.170,408.082,-156.700,173.527,50.103,160.269
C00581=1021.180,408.328,-156.745,173.538,50.104,160.272
C00582=1021.191,408.573,-156.791,173.552,50.105,160.274
C00583=1021.201,408.819,-156.837,173.564,50.107,160.277
C00584=1021.213,409.064,-156.882,173.576,50.107,160.279
C00585=1021.223,409.310,-156.929,173.589,50.109,160.281
C00586=1021.233,409.556,-156.974,173.601,50.110,160.284
C00587=1021.244,409.801,-157.021,173.614,50.111,160.286
C00588=1021.255,410.046,-157.067,173.627,50.113,160.289
C00589=1021.265,410.292,-157.113,173.640,50.114,160.291
C00590=1021.276,410.537,-157.160,173.653,50.115,160.294
C00591=1021.287,410.783,-157.205,173.665,50.117,160.296
C00592=1021.297,411.028,-157.252,173.678,50.118,160.299
C00593=1021.308,411.274,-157.299,173.691,50.119,160.301
C00594=1021.324,411.614,-157.363,173.708,50.121,160.305
C00595=1021.339,411.955,-157.427,173.726,50.122,160.308
C00596=1021.354,412.296,-157.492,173.745,50.124,160.312
C00597=1021.368,412.636,-157.557,173.762,50.126,160.315
C00598=1021.379,412.881,-157.603,173.775,50.128,160.318
C00599=1021.391,413.127,-157.650,173.788,50.129,160.321
C00600=1021.402,413.372,-157.697,173.802,50.130,160.323
C00601=1021.413,413.617,-157.743,173.815,50.132,160.326
C00602=1021.423,413.864,-157.790,173.828,50.133,160.329
C00603=1021.434,414.109,-157.837,173.841,50.134,160.331
C00604=1021.446,414.354,-157.884,173.855,50.136,160.334
C00605=1021.457,414.599,-157.931,173.868,50.137,160.336
C00606=1021.468,414.845,-157.978,173.881,50.139,160.339
C00607=1021.480,415.091,-158.025,173.895,50.140,160.342
C00608=1021.490,415.335,-158.072,173.908,50.142,160.344
C00609=1021.502,415.581,-158.119,173.922,50.144,160.347
C00610=1021.513,415.826,-158.166,173.935,50.145,160.350
C00611=1021.524,416.071,-158.214,173.948,50.147,160.352
C00612=1021.535,416.317,-158.261,173.962,50.148,160.355
C00613=1021.546,416.562,-158.309,173.976,50.150,160.358
C00614=1021.557,416.807,-158.356,173.990,50.152,160.361
C00615=1021.569,417.052,-158.404,174.003,50.153,160.364
C00616=1021.580,417.297,-158.452,174.017,50.155,160.366
C00617=1021.591,417.543,-158.499,174.030,50.157,160.369
C00618=1021.602,417.788,-158.547,174.044,50.158,160.372
C00619=1021.614,418.033,-158.595,174.059,50.160,160.375
C00620=1021.625,418.278,-158.641,174.072,50.162,160.378
C00621=1021.636,418.523,-158.690,174.085,50.163,160.380
C00622=1021.648,418.768,-158.737,174.100,50.165,160.383
C00623=1021.660,419.013,-158.785,174.114,50.167,160.386
C00624=1021.671,419.259,-158.833,174.129,50.169,160.389
C00625=1021.683,419.504,-158.881,174.142,50.170,160.392
C00626=1021.694,419.749,-158.929,174.156,50.173,160.395
C00627=1021.706,419.994,-158.977,174.171,50.174,160.398
C00628=1021.718,420.239,-159.026,174.184,50.176,160.401
C00629=1021.729,420.484,-159.074,174.199,50.178,160.404
C00630=1021.741,420.729,-159.122,174.213,50.180,160.407
C00631=1021.752,420.975,-159.170,174.228,50.182,160.410
C00632=1021.764,421.220,-159.218,174.242,50.184,160.413
C00633=1021.776,421.465,-159.267,174.256,50.186,160.416
C00634=1021.788,421.710,-159.315,174.271,50.188,160.419
C00635=1021.800,421.956,-159.364,174.285,50.190,160.422
C00636=1021.812,422.200,-159.413,174.300,50.191,160.425
C00637=1021.823,422.445,-159.461,174.315,50.193,160.428
C00638=1021.834,422.690,-159.510,174.329,50.195,160.431
C00639=1021.847,422.935,-159.559,174.344,50.198,160.434
C00640=1021.858,423.180,-159.608,174.359,50.200,160.437
C00641=1021.870,423.424,-159.656,174.373,50.201,160.440
C00642=1021.882,423.670,-159.705,174.389,50.204,160.443
C00643=1021.894,423.915,-159.754,174.403,50.205,160.446
C00644=1021.906,424.160,-159.802,174.418,50.208,160.450
C00645=1021.918,424.404,-159.852,174.432,50.210,160.453
C00646=1021.931,424.650,-159.901,174.448,50.212,160.456
C00647=1021.942,424.894,-159.950,174.463,50.214,160.459
C00648=1021.954,425.140,-159.999,174.478,50.216,160.462
C00649=1021.966,425.384,-160.048,174.493,50.219,160.465
C00650=1021.979,425.629,-160.098,174.508,50.221,160.469
C00651=1021.991,425.874,-160.147,174.523,50.223,160.472
C00652=1022.002,426.119,-160.197,174.539,50.226,160.475
C00653=1022.014,426.364,-160.246,174.554,50.228,160.478
C00654=1022.028,426.645,-160.303,174.571,50.230,160.482
C00655=1022.043,426.926,-160.360,174.589,50.233,160.486
C00656=1022.056,427.207,-160.417,174.607,50.235,160.490
C00657=1022.070,427.488,-160.474,174.625,50.238,160.494
C00658=1022.083,427.733,-160.524,174.641,50.240,160.497
C00659=1022.095,427.978,-160.574,174.656,50.243,160.500
C00660=1022.107,428.222,-160.625,174.672,50.245,160.504
C00661=1022.120,428.467,-160.674,174.688,50.247,160.507
C00662=1022.133,428.712,-160.724,174.703,50.250,160.510
C00663=1022.145,428.956,-160.774,174.719,50.252,160.514
C00664=1022.157,429.201,-160.824,174.735,50.255,160.517
C00665=1022.170,429.446,-160.874,174.751,50.258,160.521
C00666=1022.183,429.691,-160.924,174.767,50.259,160.524
C00667=1022.195,429.935,-160.975,174.783,50.262,160.528
C00668=1022.208,430.180,-161.025,174.799,50.265,160.531
C00669=1022.220,430.424,-161.075,174.815,50.268,160.535
C00670=1022.233,430.669,-161.126,174.832,50.270,160.538
C00671=1022.246,430.914,-161.176,174.848,50.272,160.542
C00672=1022.259,431.158,-161.226,174.864,50.275,160.545
C00673=1022.271,431.403,-161.276,174.880,50.278,160.549
C00674=1022.284,431.647,-161.327,174.897,50.280,160.552
C00675=1022.297,431.892,-161.378,174.913,50.283,160.556
C00676=1022.310,432.136,-161.429,174.929,50.285,160.559
C00677=1022.323,432.381,-161.479,174.946,50.288,160.563
C00678=1022.336,432.626,-161.530,174.963,50.290,160.567
C00679=1022.348,432.870,-161.581,174.980,50.293,160.570
C00680=1022.362,433.115,-161.632,174.995,50.296,160.574
C00681=1022.375,433.358,-161.683,175.013,50.299,160.578
C00682=1022.388,433.603,-161.735,175.029,50.301,160.581
C00683=1022.400,433.847,-161.785,175.046,50.304,160.585
C00684=1022.414,434.092,-161.837,175.063,50.307,160.589
C00685=1022.427,434.336,-161.888,175.080,50.310,160.593
C00686=1022.041,432.392,-161.817,174.936,50.356,160.582
C00687=1022.027,432.148,-161.767,174.920,50.353,160.578
C00688=1022.014,431.903,-161.715,174.903,50.350,160.574
C00689=1022.001,431.659,-161.665,174.887,50.348,160.571
C00690=1021.989,431.413,-161.614,174.870,50.346,160.567
C00691=1021.976,431.169,-161.563,174.853,50.343,160.564
C00692=1021.964,430.924,-161.513,174.838,50.340,160.560
C00693=1021.950,430.681,-161.463,174.821,50.338,160.556
C00694=1021.938,430.436,-161.413,174.805,50.336,160.553
C00695=1021.925,430.191,-161.362,174.789,50.333,160.550
C00696=1021.912,429.946,-161.312,174.773,50.331,160.546
C00697=1021.900,429.701,-161.262,174.756,50.329,160.543
C00698=1021.887,429.457,-161.211,174.741,50.326,160.539
C00699=1021.874,429.212,-161.161,174.724,50.324,160.536
C00700=1021.862,428.968,-161.111,174.709,50.322,160.532
C00701=1021.850,428.723,-161.061,174.692,50.319,160.529
C00702=1021.838,428.478,-161.011,174.677,50.317,160.526
C00703=1021.824,428.233,-160.961,174.662,50.315,160.522
C00704=1021.812,427.989,-160.911,174.645,50.312,160.519
C00705=1021.800,427.745,-160.862,174.630,50.310,160.515
C00706=1021.788,427.500,-160.812,174.615,50.308,160.512
C00707=1021.775,427.241,-160.759,174.598,50.305,160.509
C00708=1021.762,426.983,-160.707,174.582,50.303,160.505
C00709=1021.749,426.725,-160.655,174.565,50.301,160.502
C00710=1021.736,426.467,-160.603,174.549,50.298,160.498
C00711=1021.725,426.222,-160.553,174.534,50.297,160.495
C00712=1021.712,425.978,-160.503,174.518,50.294,160.492
C00713=1021.700,425.732,-160.454,174.503,50.292,160.489
C00714=1021.689,425.487,-160.405,174.488,50.290,160.485
C00715=1021.676,425.243,-160.354,174.473,50.288,160.482
C00716=1021.664,424.997,-160.306,174.458,50.286,160.479
C00717=1021.652,424.753,-160.257,174.443,50.283,160.476
C00718=1021.640,424.508,-160.208,174.428,50.282,160.473
C00719=1021.628,424.263,-160.159,174.413,50.279,160.469
C00720=1021.616,424.017,-160.109,174.398,50.278,160.466
C00721=1021.604,423.773,-160.061,174.382,50.275,160.463
C00722=1021.592,423.527,-160.012,174.368,50.274,160.460
C00723=1021.580,423.283,-159.963,174.353,50.272,160.457
C00724=1021.568,423.038,-159.914,174.338,50.270,160.454
C00725=1021.557,422.792,-159.866,174.323,50.268,160.451
C00726=1021.545,422.548,-159.817,174.309,50.266,160.448
C00727=1021.533,422.303,-159.768,174.294,50.264,160.445
C00728=1021.520,422.058,-159.719,174.279,50.262,160.442
C00729=1021.509,421.813,-159.671,174.264,50.260,160.439
C00730=1021.498,421.568,-159.622,174.250,50.258,160.436
C00731=1021.486,421.323,-159.574,174.236,50.256,160.432
C00732=1021.475,421.078,-159.525,174.221,50.255,160.430
C00733=1021.462,420.832,-159.477,174.207,50.253,160.427
C00734=1021.450,420.587,-159.430,174.192,50.251,160.424
C00735=1021.439,420.342,-159.381,174.178,50.249,160.421
C00736=1021.428,420.097,-159.334,174.164,50.248,160.418
C00737=1021.416,419.851,-159.285,174.149,50.246,160.415
C00738=1021.404,419.607,-159.237,174.136,50.244,160.412
C00739=1021.392,419.362,-159.189,174.121,50.243,160.409
C00740=1021.381,419.117,-159.141,174.108,50.241,160.406
C00741=1021.370,418.872,-159.093,174.093,50.239,160.403
C00742=1021.358,418.626,-159.046,174.079,50.238,160.400
C00743=1021.347,418.381,-158.998,174.066,50.236,160.398
C00744=1021.335,418.135,-158.950,174.051,50.234,160.395
C00745=1021.325,417.891,-158.902,174.037,50.232,160.392
C00746=1021.313,417.646,-158.855,174.023,50.231,160.389
C00747=1021.301,417.400,-158.808,174.010,50.230,160.386
C00748=1021.290,417.155,-158.759,173.996,50.228,160.384
C00749=1021.279,416.910,-158.712,173.983,50.226,160.381
C00750=1021.268,416.664,-158.664,173.968,50.225,160.378
C00751=1021.256,416.419,-158.617,173.955,50.223,160.375
C00752=1021.245,416.174,-158.570,173.941,50.222,160.373
C00753=1021.234,415.928,-158.522,173.928,50.220,160.370
C00754=1021.223,415.683,-158.475,173.914,50.218,160.367
C00755=1021.212,415.438,-158.428,173.900,50.217,160.364
C00756=1021.201,415.192,-158.381,173.887,50.216,160.362
C00757=1021.190,414.948,-158.333,173.873,50.214,160.359
C00758=1021.178,414.702,-158.286,173.860,50.213,160.356
C00759=1021.167,414.457,-158.240,173.847,50.212,160.354
C00760=1021.156,414.212,-158.193,173.833,50.210,160.351
C00761=1021.146,413.966,-158.145,173.820,50.209,160.348
C00762=1021.134,413.720,-158.099,173.807,50.207,160.346
C00763=1021.123,413.475,-158.052,173.794,50.206,160.343
C00764=1021.112,413.229,-158.005,173.781,50.205,160.341
C00765=1021.101,412.984,-157.959,173.767,50.203,160.338
C00766=1021.090,412.740,-157.912,173.754,50.202,160.335
C00767=1021.075,412.397,-157.847,173.736,50.201,160.332
C00768=1021.060,412.054,-157.782,173.717,50.199,160.328
C00769=1021.044,411.711,-157.717,173.700,50.197,160.325
C00770=1021.029,411.368,-157.652,173.682,50.196,160.321
C00771=1021.019,411.122,-157.606,173.669,50.195,160.319
C00772=1021.008,410.877,-157.560,173.656,50.193,160.316
C00773=1020.997,410.632,-157.514,173.643,50.192,160.314
C00774=1020.987,410.386,-157.468,173.631,50.191,160.311
C00775=1020.976,410.140,-157.420,173.618,50.190,160.309
C00776=1020.965,409.894,-157.374,173.605,50.189,160.306
C00777=1020.954,409.649,-157.328,173.592,50.187,160.304
C00778=1020.944,409.403,-157.283,173.580,50.186,160.301
C00779=1020.934,409.159,-157.236,173.567,50.185,160.299
C00780=1020.923,408.913,-157.190,173.555,50.184,160.296
C00781=1020.912,408.668,-157.144,173.542,50.183,160.294
C00782=1020.901,408.421,-157.099,173.529,50.182,160.292
C00783=1020.891,408.176,-157.053,173.517,50.181,160.289
C00784=1020.880,407.931,-157.008,173.504,50.180,160.287
C00785=1020.869,407.685,-156.962,173.492,50.179,160.285
C00786=1020.859,407.440,-156.916,173.480,50.179,160.282
C00787=1020.848,407.193,-156.871,173.467,50.177,160.280
C00788=1020.838,406.948,-156.825,173.455,50.177,160.278
C00789=1020.827,406.703,-156.780,173.442,50.176,160.275
C00790=1020.817,406.457,-156.735,173.430,50.174,160.273
C00791=1020.806,406.211,-156.689,173.418,50.174,160.271
C00792=1020.796,405.965,-156.644,173.406,50.173,160.268
C00793=1020.785,405.721,-156.599,173.394,50.172,160.266
C00794=1020.775,405.474,-156.554,173.382,50.171,160.264
C00795=1020.765,405.229,-156.508,173.370,50.170,160.262
C00796=1020.754,404.983,-156.463,173.357,50.170,160.259
C00797=1020.744,404.737,-156.418,173.346,50.169,160.257
C00798=1020.733,404.492,-156.373,173.334,50.168,160.255
C00799=1020.723,404.246,-156.328,173.321,50.167,160.252
C00800=1020.713,404.001,-156.283,173.309,50.166,160.250
C00801=1020.703,403.754,-156.238,173.298,50.166,160.248
C00802=1020.693,403.509,-156.193,173.286,50.165,160.246
C00803=1020.682,403.264,-156.148,173.274,50.164,160.244
C00804=1020.672,403.018,-156.103,173.262,50.163,160.241
C00805=1020.662,402.773,-156.058,173.251,50.163,160.239
C00806=1020.653,402.527,-156.013,173.238,50.163,160.237
C00807=1020.642,402.281,-155.968,173.226,50.162,160.235
C00808=1020.632,402.036,-155.924,173.215,50.161,160.233
C00809=1020.623,401.790,-155.880,173.203,50.160,160.231
C00810=1020.612,401.543,-155.834,173.192,50.160,160.229
C00811=1020.603,401.298,-155.790,173.181,50.159,160.226
C00812=1020.593,401.052,-155.745,173.168,50.159,160.224
C00813=1020.582,400.807,-155.700,173.157,50.158,160.222
C00814=1020.573,400.561,-155.656,173.145,50.157,160.220
C00815=1020.563,400.315,-155.611,173.134,50.157,160.218
C00816=1020.552,400.069,-155.568,173.123,50.157,160.216
C00817=1020.543,399.823,-155.523,173.111,50.156,160.214
C00818=1020.533,399.577,-155.479,173.100,50.155,160.212
C00819=1020.523,399.332,-155.435,173.088,50.155,160.210
C00820=1020.513,399.086,-155.390,173.077,50.154,160.208
C00821=1020.503,398.841,-155.346,173.066,50.154,160.206
C00822=1020.494,398.595,-155.302,173.054,50.154,160.204
C00823=1020.484,398.349,-155.258,173.043,50.153,160.202
C00824=1020.474,398.103,-155.214,173.032,50.153,160.200
C00825=1020.464,397.857,-155.170,173.021,50.152,160.198
C00826=1020.454,397.611,-155.126,173.009,50.152,160.196
C00827=1020.441,397.291,-155.068,172.994,50.151,160.193
C00828=1020.429,396.971,-155.013,172.981,50.151,160.191
C00829=1020.416,396.651,-154.955,172.965,50.151,160.188
C00830=1020.403,396.330,-154.898,172.952,50.150,160.186
C00831=1020.393,396.084,-154.854,172.941,50.150,160.184
C00832=1020.384,395.839,-154.812,172.929,50.149,160.182
C00833=1020.374,395.593,-154.768,172.918,50.150,160.180
C00834=1020.365,395.347,-154.724,172.907,50.149,160.178
C00835=1020.356,395.130,-154.687,172.898,50.149,160.176
C00836=1020.348,394.915,-154.648,172.889,50.149,160.175
C00837=1020.340,394.699,-154.610,172.879,50.149,160.173
C00838=1020.331,394.483,-154.572,172.869,50.149,160.171
C00839=1020.322,394.267,-154.533,172.860,50.148,160.170
C00840=1020.315,394.051,-154.496,172.850,50.148,160.168
C00841=1020.306,393.835,-154.458,172.840,50.148,160.166
C00842=1020.298,393.620,-154.419,172.831,50.148,160.165
C00843=1020.288,393.373,-154.377,172.821,50.148,160.163
C00844=1020.278,393.127,-154.332,172.809,50.148,160.161
C00845=1020.269,392.881,-154.290,172.799,50.147,160.159
C00846=1020.259,392.635,-154.247,172.788,50.148,160.157
C00847=1020.251,392.390,-154.204,172.778,50.148,160.156
C00848=1020.241,392.143,-154.161,172.768,50.148,160.154
C00849=1020.231,391.897,-154.118,172.756,50.147,160.152
C00850=1020.222,391.651,-154.075,172.745,50.147,160.150
C00851=1020.212,391.404,-154.032,172.735,50.147,160.148
C00852=1020.203,391.158,-153.990,172.725,50.147,160.147
C00853=1020.193,390.912,-153.947,172.715,50.147,160.145
C00854=1020.184,390.667,-153.904,172.704,50.147,160.143
C00855=1020.175,390.421,-153.861,172.693,50.147,160.141
C00856=1020.166,390.174,-153.819,172.683,50.148,160.140
C00857=1020.157,389.928,-153.776,172.672,50.148,160.138
C00858=1020.147,389.682,-153.733,172.662,50.148,160.136
C00859=1020.138,389.436,-153.691,172.652,50.148,160.134
C00860=1020.128,389.190,-153.649,172.642,50.148,160.133
C00861=1020.119,388.943,-153.605,172.631,50.148,160.131
C00862=1020.110,388.698,-153.563,172.621,50.148,160.129
C00863=1020.101,388.451,-153.521,172.610,50.148,160.128
C00864=1020.092,388.205,-153.479,172.601,50.149,160.126
C00865=1020.082,387.959,-153.436,172.590,50.149,160.124
C00866=1020.073,387.713,-153.394,172.580,50.149,160.123
C00867=1020.064,387.467,-153.352,172.569,50.149,160.121
C00868=1020.055,387.221,-153.310,172.559,50.149,160.119
C00869=1020.046,386.974,-153.266,172.550,50.149,160.118
C00870=1020.037,386.727,-153.225,172.539,50.150,160.116
C00871=1020.028,386.482,-153.182,172.529,50.150,160.114
C00872=1020.019,386.235,-153.141,172.519,50.151,160.113
C00873=1020.010,385.989,-153.099,172.509,50.150,160.111
C00874=1020.000,385.743,-153.056,172.499,50.151,160.110
C00875=1019.991,385.497,-153.015,172.489,50.152,160.108
C00876=1019.983,385.250,-152.973,172.479,50.151,160.106
C00877=1019.974,385.004,-152.931,172.469,50.152,160.105
C00878=1019.963,384.757,-152.890,172.459,50.152,160.103
C00879=1019.954,384.511,-152.848,172.449,50.153,160.102
C00880=1019.945,384.265,-152.806,172.440,50.153,160.100
C00881=1019.937,384.018,-152.765,172.429,50.154,160.099
C00882=1019.928,383.772,-152.723,172.420,50.154,160.097
C00883=1019.918,383.526,-152.682,172.410,50.155,160.096
C00884=1019.909,383.279,-152.640,172.400,50.155,160.094
C00885=1019.901,383.034,-152.599,172.390,50.156,160.093
C00886=1019.892,382.787,-152.557,172.381,50.156,160.091
C00887=1019.879,382.444,-152.499,172.366,50.157,160.089
C00888=1019.867,382.101,-152.442,172.353,50.157,160.087
C00889=1019.855,381.758,-152.385,172.341,50.158,160.085
C00890=1019.842,381.415,-152.327,172.326,50.159,160.083
C00891=1019.833,381.169,-152.285,172.317,50.160,160.081
C00892=1019.825,380.923,-152.245,172.308,50.160,160.080
C00893=1019.816,380.676,-152.203,172.298,50.160,160.078
C00894=1019.806,380.430,-152.163,172.288,50.162,160.077
C00895=1019.797,380.183,-152.121,172.278,50.162,160.075
C00896=1019.789,379.937,-152.080,172.269,50.162,160.074
C00897=1019.780,379.691,-152.039,172.260,50.163,160.073
C00898=1019.772,379.444,-151.998,172.250,50.164,160.071
C00899=1019.763,379.198,-151.957,172.241,50.165,160.070
C00900=1019.754,378.951,-151.916,172.231,50.165,160.068
C00901=1019.745,378.704,-151.875,172.222,50.166,160.067
C00902=1019.737,378.458,-151.834,172.213,50.166,160.066
C00903=1019.729,378.212,-151.792,172.204,50.167,160.064
C00904=1019.720,377.966,-151.752,172.194,50.168,160.063
C00905=1019.711,377.719,-151.711,172.185,50.169,160.061
C00906=1019.703,377.472,-151.671,172.175,50.169,160.060
C00907=1019.694,377.225,-151.630,172.166,50.170,160.059
C00908=1019.686,376.980,-151.588,172.157,50.171,160.057
C00909=1019.677,376.733,-151.548,172.148,50.171,160.056
C00910=1019.669,376.487,-151.507,172.138,50.172,160.055
C00911=1019.660,376.240,-151.466,172.129,50.173,160.053
C00912=1019.652,375.994,-151.426,172.120,50.174,160.052
C00913=1019.643,375.747,-151.385,172.111,50.175,160.051
C00914=1019.635,375.500,-151.345,172.102,50.176,160.049
C00915=1019.626,375.253,-151.305,172.093,50.177,160.048
C00916=1019.618,375.007,-151.264,172.083,50.177,160.047
C00917=1019.609,374.761,-151.224,172.074,50.178,160.045
C00918=1019.600,374.514,-151.185,172.065,50.180,160.044
C00919=1019.592,374.267,-151.144,172.056,50.181,160.043
C00920=1019.583,374.021,-151.104,172.047,50.182,160.042
C00921=1019.575,373.774,-151.064,172.038,50.183,160.040
C00922=1019.566,373.528,-151.024,172.029,50.184,160.039
C00923=1019.558,373.281,-150.984,172.019,50.185,160.038
C00924=1019.549,373.034,-150.943,172.010,50.186,160.036
C00925=1019.541,372.787,-150.903,172.001,50.186,160.035
C00926=1019.532,372.541,-150.863,171.992,50.188,160.034
C00927=1019.525,372.295,-150.823,171.984,50.189,160.033
C00928=1019.515,372.048,-150.783,171.975,50.190,160.031
C00929=1019.507,371.801,-150.744,171.966,50.191,160.030
C00930=1019.499,371.554,-150.704,171.957,50.192,160.029
C00931=1019.490,371.308,-150.664,171.948,50.193,160.028
C00932=1019.483,371.061,-150.624,171.939,50.194,160.027
C00933=1019.474,370.815,-150.584,171.931,50.195,160.026
C00934=1019.466,370.567,-150.544,171.922,50.196,160.024
C00935=1019.457,370.321,-150.504,171.913,50.198,160.023
C00936=1019.449,370.074,-150.464,171.904,50.199,160.022
C00937=1019.441,369.828,-150.425,171.895,50.200,160.021
C00938=1019.433,369.581,-150.385,171.887,50.201,160.020
C00939=1019.425,369.334,-150.346,171.878,50.202,160.018
C00940=1019.416,369.088,-150.306,171.869,50.203,160.017
C00941=1019.409,368.841,-150.266,171.860,50.205,160.016
C00942=1019.400,368.594,-150.227,171.852,50.205,160.015
C00943=1019.392,368.347,-150.187,171.843,50.207,160.014
C00944=1019.384,368.101,-150.148,171.835,50.208,160.013
C00945=1019.376,367.854,-150.108,171.826,50.209,160.011
C00946=1019.368,367.607,-150.069,171.818,50.211,160.010
C00947=1019.359,367.347,-150.028,171.809,50.212,160.009
C00948=1019.351,367.087,-149.986,171.799,50.213,160.008
C00949=1019.342,366.826,-149.945,171.790,50.215,160.007
C00950=1019.333,366.565,-149.903,171.781,50.217,160.006
C00951=1019.325,366.318,-149.864,171.772,50.218,160.005
C00952=1019.317,366.071,-149.825,171.765,50.219,160.004
C00953=1019.309,365.825,-149.786,171.756,50.221,160.003
C00954=1019.301,365.578,-149.748,171.747,50.222,160.001
C00955=1019.292,365.332,-149.708,171.739,50.223,160.000
C00956=1019.284,365.085,-149.669,171.730,50.225,159.999
C00957=1019.276,364.838,-149.630,171.722,50.227,159.998
C00958=1019.268,364.590,-149.591,171.714,50.228,159.997
C00959=1019.260,364.344,-149.552,171.705,50.229,159.996
C00960=1019.252,364.097,-149.514,171.697,50.231,159.995
C00961=1019.244,363.851,-149.474,171.689,50.232,159.994
C00962=1019.236,363.603,-149.436,171.680,50.234,159.993
C00963=1019.228,363.357,-149.397,171.672,50.235,159.992
C00964=1019.220,363.110,-149.358,171.663,50.236,159.991
C00965=1019.211,362.863,-149.320,171.655,50.239,159.990
C00966=1019.204,362.616,-149.281,171.647,50.240,159.989
C00967=1019.196,362.369,-149.242,171.638,50.241,159.988
C00968=1019.188,362.122,-149.203,171.631,50.243,159.987
C00969=1019.180,361.876,-149.165,171.622,50.245,159.986
C00970=1019.172,361.629,-149.126,171.614,50.246,159.985
C00971=1019.165,361.382,-149.088,171.606,50.247,159.984
C00972=1019.157,361.135,-149.049,171.598,50.249,159.983
C00973=1019.149,360.888,-149.011,171.589,50.251,159.982
C00974=1019.141,360.641,-148.972,171.581,50.252,159.981
C00975=1019.134,360.394,-148.933,171.573,50.254,159.980
C00976=1019.126,360.147,-148.895,171.564,50.256,159.979
C00977=1019.118,359.901,-148.857,171.557,50.257,159.978
C00978=1019.110,359.653,-148.818,171.548,50.259,159.977
C00979=1019.103,359.407,-148.780,171.541,50.261,159.976
C00980=1019.095,359.160,-148.741,171.532,50.262,159.975
C00981=1019.087,358.912,-148.704,171.525,50.264,159.974
C00982=1019.078,358.666,-148.666,171.516,50.266,159.973
C00983=1019.071,358.419,-148.627,171.509,50.268,159.972
C00984=1019.063,358.171,-148.589,171.500,50.270,159.972
C00985=1019.055,357.925,-148.551,171.493,50.272,159.971
C00986=1019.047,357.678,-148.513,171.484,50.273,159.970
C00987=1019.040,357.430,-148.475,171.477,50.275,159.969
C00988=1019.033,357.184,-148.437,171.469,50.277,159.968
C00989=1019.024,356.936,-148.399,171.461,50.279,159.967
C00990=1019.016,356.690,-148.361,171.453,50.280,159.966
C00991=1019.009,356.443,-148.324,171.445,50.282,159.965
C00992=1019.001,356.195,-148.285,171.437,50.284,159.964
C00993=1018.993,355.949,-148.248,171.429,50.286,159.964
C00994=1018.985,355.702,-148.210,171.421,50.288,159.963
C00995=1018.978,355.454,-148.172,171.413,50.290,159.962
C00996=1018.970,355.207,-148.135,171.406,50.292,159.961
C00997=1018.963,354.961,-148.096,171.398,50.294,159.960
C00998=1018.955,354.714,-148.059,171.390,50.296,159.959
C00999=1018.948,354.467,-148.022,171.382,50.298,159.959
C01000=1018.939,354.219,-147.983,171.374,50.300,159.958
C01001=1018.932,353.972,-147.946,171.367,50.302,159.957
C01002=1018.924,353.726,-147.909,171.359,50.303,159.956
C01003=1018.917,353.478,-147.871,171.351,50.306,159.955
C01004=1018.910,353.231,-147.834,171.344,50.307,159.954
C01005=1018.901,352.984,-147.796,171.335,50.310,159.954
C01006=1018.894,352.737,-147.759,171.328,50.312,159.953
C01007=1018.886,352.483,-147.720,171.320,50.314,159.952
C01008=1018.879,352.231,-147.682,171.312,50.316,159.951
C01009=1018.870,351.978,-147.645,171.304,50.318,159.950
C01010=1018.862,351.725,-147.606,171.297,50.321,159.950
C01011=1018.855,351.478,-147.569,171.288,50.323,159.949
C01012=1018.847,351.231,-147.532,171.281,50.325,159.948
C01013=1018.840,350.984,-147.494,171.274,50.327,159.947
C01014=1018.833,350.737,-147.457,171.266,50.329,159.947
C01015=1018.825,350.489,-147.420,171.258,50.331,159.946
C01016=1018.818,350.242,-147.383,171.251,50.333,159.945
C01017=1018.810,349.995,-147.346,171.243,50.336,159.944
C01018=1018.803,349.748,-147.308,171.236,50.338,159.944
C01019=1018.796,349.500,-147.272,171.228,50.340,159.943
C01020=1018.788,349.253,-147.235,171.220,50.342,159.942
C01021=1018.780,349.006,-147.197,171.213,50.344,159.941
C01022=1018.772,348.759,-147.160,171.206,50.346,159.941
C01023=1018.765,348.512,-147.123,171.199,50.349,159.940
C01024=1018.758,348.265,-147.087,171.191,50.351,159.939
C01025=1018.751,348.017,-147.050,171.183,50.353,159.938
C01026=1018.743,347.770,-147.013,171.176,50.356,159.938
C01027=1018.736,347.523,-146.976,171.168,50.358,159.937
C01028=1018.728,347.276,-146.939,171.161,50.360,159.936
C01029=1018.721,347.029,-146.903,171.154,50.363,159.936
C01030=1018.713,346.782,-146.866,171.146,50.365,159.935
C01031=1018.706,346.534,-146.829,171.138,50.367,159.934
C01032=1018.698,346.287,-146.792,171.131,50.370,159.934
C01033=1018.691,346.041,-146.756,171.124,50.372,159.933
C01034=1018.684,345.793,-146.719,171.117,50.375,159.933
C01035=1018.677,345.545,-146.683,171.109,50.377,159.932
C01036=1018.669,345.298,-146.646,171.102,50.379,159.931
C01037=1018.662,345.051,-146.610,171.095,50.382,159.930
C01038=1018.655,344.804,-146.573,171.088,50.384,159.930
C01039=1018.647,344.557,-146.537,171.080,50.387,159.929
C01040=1018.640,344.309,-146.500,171.073,50.389,159.929
C01041=1018.633,344.063,-146.464,171.066,50.392,159.928
C01042=1018.625,343.815,-146.428,171.059,50.394,159.927
C01043=1018.618,343.567,-146.391,171.051,50.397,159.927
C01044=1018.611,343.321,-146.355,171.044,50.399,159.926
C01045=1018.603,343.073,-146.319,171.037,50.402,159.925
C01046=1018.596,342.826,-146.283,171.030,50.404,159.925
C01047=1018.589,342.579,-146.246,171.023,50.407,159.924
C01048=1018.582,342.331,-146.210,171.015,50.410,159.924
C01049=1018.574,342.084,-146.174,171.008,50.412,159.923
C01050=1018.567,341.837,-146.138,171.001,50.414,159.922
C01051=1018.560,341.589,-146.101,170.994,50.417,159.922
C01052=1018.553,341.342,-146.066,170.987,50.419,159.921
C01053=1018.546,341.095,-146.030,170.979,50.423,159.921
C01054=1018.539,340.848,-145.994,170.972,50.425,159.920
C01055=1018.532,340.600,-145.957,170.965,50.428,159.919
C01056=1018.524,340.353,-145.921,170.958,50.430,159.919
C01057=1018.517,340.105,-145.886,170.951,50.433,159.918
C01058=1018.510,339.859,-145.850,170.944,50.436,159.918
C01059=1018.502,339.611,-145.814,170.936,50.438,159.917
C01060=1018.496,339.363,-145.778,170.929,50.441,159.916
C01061=1018.489,339.116,-145.742,170.923,50.444,159.916
C01062=1018.482,338.869,-145.706,170.916,50.446,159.916
C01063=1018.474,338.621,-145.670,170.909,50.449,159.915
C01064=1018.467,338.374,-145.634,170.902,50.452,159.915
C01065=1018.460,338.126,-145.599,170.894,50.455,159.914
C01066=1018.453,337.880,-145.563,170.887,50.458,159.913
C01067=1018.445,337.624,-145.526,170.881,50.461,159.913
C01068=1018.438,337.368,-145.490,170.873,50.464,159.912
C01069=1018.430,337.112,-145.453,170.866,50.467,159.912
C01070=1018.423,336.856,-145.416,170.859,50.469,159.911
C01071=1018.417,336.609,-145.381,170.852,50.472,159.911
C01072=1018.409,336.361,-145.345,170.844,50.475,159.910
C01073=1018.402,336.114,-145.309,170.838,50.478,159.910
C01074=1018.395,335.867,-145.275,170.831,50.481,159.909
C01075=1018.387,335.619,-145.239,170.824,50.484,159.909
C01076=1018.380,335.372,-145.204,170.818,50.487,159.908
C01077=1018.373,335.125,-145.168,170.811,50.490,159.908
C01078=1018.367,334.877,-145.133,170.804,50.492,159.907
C01079=1018.359,334.629,-145.098,170.797,50.495,159.907
C01080=1018.352,334.382,-145.062,170.790,50.499,159.907
C01081=1018.345,334.135,-145.027,170.783,50.502,159.906
C01082=1018.339,333.888,-144.992,170.776,50.504,159.905
C01083=1018.331,333.640,-144.956,170.769,50.507,159.905
C01084=1018.325,333.392,-144.921,170.763,50.510,159.905
C01085=1018.318,333.145,-144.886,170.756,50.513,159.904
C01086=1018.311,332.898,-144.851,170.749,50.516,159.904
C01087=1018.304,332.650,-144.816,170.742,50.519,159.903
C01088=1018.297,332.403,-144.781,170.736,50.522,159.903
C01089=1018.290,332.156,-144.746,170.729,50.525,159.902
C01090=1018.283,331.908,-144.710,170.723,50.528,159.902
C01091=1018.276,331.660,-144.675,170.715,50.532,159.902
C01092=1018.269,331.413,-144.640,170.708,50.535,159.901
C01093=1018.262,331.165,-144.606,170.702,50.538,159.901
C01094=1018.255,330.918,-144.571,170.695,50.541,159.900
C01095=1018.248,330.671,-144.536,170.688,50.544,159.900
C01096=1018.241,330.424,-144.502,170.682,50.547,159.900
C01097=1018.234,330.176,-144.467,170.676,50.551,159.899
C01098=1018.228,329.928,-144.432,170.669,50.554,159.899
C01099=1018.220,329.681,-144.397,170.662,50.557,159.899
C01100=1018.214,329.433,-144.363,170.656,50.560,159.898
C01101=1018.207,329.186,-144.328,170.649,50.563,159.898
C01102=1018.200,328.938,-144.293,170.642,50.566,159.897
C01103=1018.193,328.691,-144.259,170.635,50.570,159.897
C01104=1018.186,328.443,-144.224,170.629,50.573,159.897
C01105=1018.179,328.196,-144.189,170.622,50.576,159.896
C01106=1018.172,327.948,-144.155,170.615,50.580,159.896
C01107=1018.165,327.701,-144.120,170.609,50.583,159.895
C01108=1018.159,327.453,-144.085,170.602,50.586,159.895
C01109=1018.151,327.206,-144.051,170.596,50.589,159.895
C01110=1018.145,326.958,-144.016,170.589,50.593,159.894
C01111=1018.138,326.711,-143.981,170.583,50.596,159.894
C01112=1018.132,326.463,-143.947,170.576,50.599,159.894
C01113=1018.125,326.216,-143.913,170.570,50.602,159.893
C01114=1018.118,325.969,-143.879,170.563,50.606,159.893
C01115=1018.111,325.721,-143.844,170.557,50.609,159.893
C01116=1018.104,325.473,-143.811,170.551,50.613,159.893
C01117=1018.097,325.225,-143.777,170.544,50.616,159.892
C01118=1018.090,324.978,-143.743,170.538,50.620,159.892
C01119=1018.083,324.730,-143.709,170.530,50.624,159.892
C01120=1018.076,324.483,-143.674,170.524,50.627,159.891
C01121=1018.069,324.236,-143.641,170.518,50.631,159.891
C01122=1018.062,323.988,-143.607,170.511,50.634,159.891
C01123=1018.055,323.740,-143.572,170.505,50.638,159.890
C01124=1018.048,323.492,-143.538,170.498,50.641,159.890
C01125=1018.041,323.245,-143.505,170.492,50.644,159.890
C01126=1018.034,322.998,-143.471,170.486,50.648,159.890
C01127=1018.027,322.737,-143.436,170.479,50.652,159.889
C01128=1018.020,322.477,-143.400,170.472,50.656,159.889
C01129=1018.013,322.217,-143.364,170.466,50.660,159.889
C01130=1018.006,321.957,-143.329,170.458,50.663,159.888
C01131=1017.999,321.709,-143.296,170.452,50.667,159.888
C01132=1017.992,321.461,-143.261,170.446,50.671,159.888
C01133=1017.986,321.214,-143.228,170.440,50.674,159.888
C01134=1017.978,320.966,-143.194,170.433,50.678,159.888
C01135=1017.971,320.719,-143.160,170.427,50.681,159.887
C01136=1017.965,320.471,-143.126,170.420,50.685,159.887
C01137=1017.958,320.223,-143.093,170.414,50.689,159.887
C01138=1017.952,319.976,-143.059,170.408,50.692,159.887
C01139=1017.945,319.728,-143.026,170.402,50.696,159.886
C01140=1017.938,319.480,-142.991,170.395,50.700,159.886
C01141=1017.932,319.233,-142.958,170.389,50.704,159.886
C01142=1017.925,318.985,-142.925,170.383,50.707,159.886
C01143=1017.918,318.738,-142.891,170.377,50.711,159.886
C01144=1017.912,318.490,-142.857,170.371,50.715,159.885
C01145=1017.905,318.243,-142.824,170.364,50.719,159.885
C01146=1017.898,317.995,-142.790,170.358,50.722,159.885
C01147=1017.892,317.747,-142.757,170.352,50.726,159.885
C01148=1017.885,317.500,-142.724,170.346,50.730,159.885
C01149=1017.879,317.252,-142.689,170.339,50.734,159.884
C01150=1017.872,317.004,-142.656,170.333,50.737,159.884
C01151=1017.865,316.757,-142.623,170.327,50.741,159.884
C01152=1017.858,316.509,-142.590,170.321,50.745,159.884
C01153=1017.853,316.262,-142.556,170.314,50.749,159.884
C01154=1017.846,316.013,-142.523,170.308,50.752,159.883
C01155=1017.839,315.766,-142.489,170.302,50.757,159.883
C01156=1017.832,315.518,-142.456,170.296,50.761,159.883
C01157=1017.826,315.271,-142.423,170.290,50.764,159.883
C01158=1017.820,315.023,-142.389,170.284,50.768,159.883
C01159=1017.813,314.775,-142.356,170.277,50.772,159.883
C01160=1017.806,314.528,-142.323,170.271,50.776,159.882
C01161=1017.800,314.280,-142.290,170.265,50.780,159.882
C01162=1017.794,314.032,-142.256,170.259,50.784,159.882
C01163=1017.787,313.785,-142.223,170.253,50.787,159.882
C01164=1017.781,313.537,-142.190,170.247,50.792,159.882
C01165=1017.774,313.289,-142.156,170.241,50.796,159.882
C01166=1017.768,313.042,-142.124,170.235,50.799,159.881
C01167=1017.762,312.794,-142.090,170.228,50.803,159.881
C01168=1017.756,312.546,-142.057,170.222,50.808,159.881
C01169=1017.749,312.299,-142.024,170.217,50.811,159.881
C01170=1017.742,312.051,-141.991,170.211,50.815,159.881
C01171=1017.736,311.803,-141.958,170.205,50.819,159.881
C01172=1017.730,311.556,-141.925,170.199,50.823,159.881
C01173=1017.724,311.308,-141.892,170.193,50.827,159.881
C01174=1017.717,311.060,-141.858,170.187,50.831,159.880
C01175=1017.711,310.813,-141.825,170.181,50.835,159.880
C01176=1017.704,310.565,-141.793,170.175,50.839,159.880
C01177=1017.699,310.317,-141.759,170.169,50.843,159.880
C01178=1017.693,310.070,-141.727,170.163,50.847,159.880
C01179=1017.686,309.822,-141.694,170.156,50.851,159.880
C01180=1017.680,309.574,-141.661,170.151,50.856,159.880
C01181=1017.673,309.326,-141.628,170.145,50.860,159.880
C01182=1017.666,309.079,-141.596,170.139,50.864,159.880
C01183=1017.660,308.831,-141.563,170.133,50.868,159.880
C01184=1017.653,308.583,-141.532,170.127,50.873,159.880
C01185=1017.647,308.336,-141.499,170.121,50.877,159.880
C01186=1017.640,308.088,-141.467,170.115,50.881,159.880
C01187=1017.633,307.833,-141.433,170.109,50.886,159.880
C01188=1017.627,307.579,-141.400,170.104,50.890,159.880
C01189=1017.619,307.324,-141.367,170.096,50.894,159.879
C01190=1017.613,307.070,-141.334,170.090,50.899,159.879
C01191=1017.607,306.821,-141.302,170.085,50.903,159.879
C01192=1017.599,306.573,-141.269,170.079,50.908,159.879
C01193=1017.593,306.325,-141.237,170.073,50.912,159.879
C01194=1017.586,306.078,-141.205,170.067,50.917,159.879
C01195=1017.580,305.830,-141.173,170.061,50.921,159.879
C01196=1017.573,305.582,-141.141,170.055,50.925,159.879
C01197=1017.567,305.334,-141.109,170.050,50.930,159.879
C01198=1017.561,305.087,-141.076,170.044,50.934,159.879
C01199=1017.554,304.839,-141.045,170.038,50.939,159.879
C01200=1017.548,304.591,-141.012,170.032,50.943,159.879
C01201=1017.541,304.343,-140.981,170.026,50.948,159.879
C01202=1017.535,304.096,-140.948,170.020,50.952,159.879
C01203=1017.528,303.848,-140.916,170.015,50.956,159.879
C01204=1017.522,303.599,-140.884,170.009,50.961,159.879
C01205=1017.516,303.352,-140.852,170.003,50.965,159.879
C01206=1017.509,303.104,-140.820,169.997,50.970,159.879
C01207=1017.503,302.856,-140.788,169.991,50.974,159.879
C01208=1017.496,302.608,-140.756,169.986,50.979,159.879
C01209=1017.490,302.360,-140.724,169.980,50.984,159.879
C01210=1017.484,302.113,-140.693,169.974,50.988,159.879
C01211=1017.478,301.865,-140.660,169.968,50.993,159.879
C01212=1017.471,301.618,-140.629,169.963,50.997,159.879
C01213=1017.465,301.369,-140.597,169.957,51.001,159.879
C01214=1017.459,301.121,-140.565,169.951,51.006,159.879
C01215=1017.452,300.873,-140.533,169.945,51.011,159.879
C01216=1017.446,300.626,-140.501,169.940,51.015,159.879
C01217=1017.440,300.378,-140.470,169.934,51.020,159.879
C01218=1017.434,300.130,-140.437,169.928,51.025,159.880
C01219=1017.427,299.882,-140.406,169.922,51.029,159.880
C01220=1017.421,299.634,-140.374,169.917,51.034,159.880
C01221=1017.415,299.386,-140.343,169.911,51.038,159.880
C01222=1017.409,299.139,-140.311,169.905,51.043,159.880
C01223=1017.403,298.891,-140.278,169.900,51.048,159.880
C01224=1017.396,298.643,-140.247,169.894,51.052,159.880
C01225=1017.390,298.395,-140.215,169.888,51.057,159.880
C01226=1017.384,298.148,-140.184,169.882,51.062,159.880
C01227=1017.378,297.900,-140.152,169.877,51.067,159.880
C01228=1017.371,297.652,-140.120,169.871,51.071,159.880
C01229=1017.365,297.403,-140.088,169.865,51.076,159.880
C01230=1017.359,297.156,-140.057,169.860,51.081,159.880
C01231=1017.353,296.908,-140.025,169.854,51.085,159.880
C01232=1017.347,296.659,-139.994,169.850,51.090,159.881
C01233=1017.341,296.412,-139.963,169.844,51.094,159.881
C01234=1017.335,296.164,-139.931,169.838,51.100,159.881
C01235=1017.329,295.916,-139.899,169.833,51.104,159.881
C01236=1017.323,295.668,-139.868,169.827,51.109,159.881
C01237=1017.317,295.420,-139.836,169.821,51.114,159.881
C01238=1017.311,295.172,-139.804,169.816,51.119,159.881
C01239=1017.304,294.925,-139.773,169.810,51.123,159.881
C01240=1017.299,294.676,-139.742,169.805,51.128,159.881
C01241=1017.293,294.429,-139.711,169.799,51.133,159.881
C01242=1017.287,294.181,-139.679,169.793,51.138,159.881
C01243=1017.281,293.939,-139.648,169.788,51.143,159.882
C01244=1017.275,293.695,-139.617,169.782,51.147,159.882
C01245=1017.269,293.454,-139.587,169.778,51.152,159.882
C01246=1017.263,293.212,-139.556,169.772,51.157,159.882
C01247=1017.257,292.968,-139.525,169.767,51.162,159.882
C01248=1017.251,292.727,-139.495,169.761,51.166,159.882
C01249=1017.246,292.484,-139.464,169.755,51.171,159.882
C01250=1017.240,292.242,-139.434,169.750,51.176,159.882
C01251=1017.233,291.993,-139.403,169.744,51.182,159.883
C01252=1017.227,291.746,-139.372,169.739,51.187,159.883
C01253=1017.221,291.498,-139.341,169.733,51.191,159.883
C01254=1017.214,291.250,-139.310,169.728,51.196,159.883
C01255=1017.209,291.002,-139.279,169.722,51.201,159.883
C01256=1017.203,290.754,-139.249,169.717,51.207,159.883
C01257=1017.196,290.506,-139.217,169.712,51.212,159.884
C01258=1017.190,290.258,-139.187,169.706,51.217,159.884
C01259=1017.184,290.010,-139.156,169.701,51.222,159.884
C01260=1017.178,289.762,-139.125,169.695,51.227,159.884
C01261=1017.172,289.514,-139.094,169.690,51.232,159.884
C01262=1017.166,289.266,-139.064,169.684,51.237,159.885
C01263=1017.159,289.018,-139.033,169.679,51.242,159.885
C01264=1017.153,288.770,-139.002,169.674,51.248,159.885
C01265=1017.147,288.522,-138.971,169.668,51.253,159.885
C01266=1017.141,288.274,-138.941,169.663,51.258,159.885
C01267=1017.135,288.026,-138.911,169.657,51.263,159.885
C01268=1017.128,287.778,-138.879,169.652,51.268,159.886
C01269=1017.123,287.530,-138.849,169.647,51.274,159.886
C01270=1017.116,287.282,-138.818,169.642,51.279,159.886
C01271=1017.110,287.034,-138.788,169.636,51.284,159.886
C01272=1017.104,286.786,-138.758,169.631,51.289,159.887
C01273=1017.098,286.538,-138.727,169.625,51.294,159.887
C01274=1017.092,286.290,-138.696,169.620,51.300,159.887
C01275=1017.086,286.042,-138.666,169.615,51.305,159.887
C01276=1017.080,285.794,-138.635,169.610,51.311,159.888
C01277=1017.074,285.546,-138.605,169.604,51.316,159.888
C01278=1017.068,285.298,-138.575,169.598,51.321,159.888
C01279=1017.062,285.049,-138.544,169.593,51.327,159.888
C01280=1017.056,284.802,-138.514,169.587,51.332,159.888
C01281=1017.050,284.554,-138.483,169.582,51.337,159.889
C01282=1017.044,284.305,-138.453,169.577,51.343,159.889
C01283=1017.038,284.057,-138.422,169.571,51.348,159.889
C01284=1017.032,283.810,-138.392,169.566,51.354,159.890
C01285=1017.025,283.561,-138.362,169.561,51.359,159.890
C01286=1017.020,283.313,-138.332,169.556,51.364,159.890
C01287=1017.014,283.065,-138.302,169.551,51.370,159.890
C01288=1017.007,282.818,-138.272,169.545,51.375,159.891
C01289=1017.001,282.569,-138.241,169.540,51.381,159.891
C01290=1016.995,282.321,-138.212,169.534,51.387,159.891
C01291=1016.989,282.073,-138.181,169.529,51.392,159.891
C01292=1016.983,281.825,-138.152,169.523,51.398,159.892
C01293=1016.977,281.576,-138.122,169.518,51.403,159.892
C01294=1016.971,281.328,-138.091,169.513,51.409,159.892
C01295=1016.965,281.080,-138.061,169.508,51.414,159.893
C01296=1016.959,280.832,-138.032,169.503,51.420,159.893
C01297=1016.953,280.585,-138.001,169.498,51.425,159.893
C01298=1016.947,280.336,-137.971,169.493,51.431,159.894
C01299=1016.941,280.088,-137.941,169.487,51.436,159.894
C01300=1016.935,279.840,-137.911,169.482,51.442,159.894
C01301=1016.929,279.592,-137.882,169.476,51.448,159.894
C01302=1016.923,279.344,-137.851,169.471,51.454,159.895
C01303=1016.917,279.108,-137.823,169.467,51.459,159.895
C01304=1016.911,278.872,-137.795,169.461,51.464,159.895
C01305=1016.906,278.635,-137.766,169.456,51.470,159.896
C01306=1016.900,278.399,-137.738,169.451,51.475,159.896
C01307=1016.895,278.162,-137.709,169.447,51.481,159.896
C01308=1016.889,277.926,-137.681,169.442,51.486,159.897
C01309=1016.883,277.690,-137.652,169.437,51.492,159.897
C01310=1016.878,277.454,-137.623,169.431,51.497,159.897
C01311=1016.872,277.206,-137.594,169.426,51.503,159.898
C01312=1016.866,276.957,-137.565,169.421,51.508,159.898
C01313=1016.861,276.709,-137.534,169.416,51.514,159.898
C01314=1016.855,276.461,-137.505,169.411,51.519,159.898
C01315=1016.848,276.213,-137.475,169.406,51.525,159.899
C01316=1016.843,275.965,-137.445,169.401,51.531,159.899
C01317=1016.837,275.717,-137.416,169.396,51.537,159.900
C01318=1016.831,275.468,-137.387,169.390,51.543,159.900
C01319=1016.825,275.221,-137.357,169.385,51.549,159.900
C01320=1016.819,274.972,-137.327,169.380,51.555,159.901
C01321=1016.813,274.724,-137.298,169.375,51.561,159.901
C01322=1016.807,274.476,-137.269,169.370,51.567,159.902
C01323=1016.801,274.228,-137.240,169.365,51.572,159.902
C01324=1016.795,273.980,-137.210,169.359,51.579,159.902
C01325=1016.789,273.732,-137.180,169.354,51.585,159.903
C01326=1016.783,273.484,-137.151,169.349,51.590,159.903
C01327=1016.777,273.235,-137.121,169.344,51.596,159.903
C01328=1016.771,272.987,-137.092,169.339,51.602,159.904
C01329=1016.766,272.739,-137.063,169.334,51.608,159.904
C01330=1016.759,272.490,-137.034,169.329,51.614,159.905
C01331=1016.754,272.242,-137.004,169.323,51.620,159.905
C01332=1016.747,271.994,-136.975,169.319,51.627,159.905
C01333=1016.742,271.745,-136.945,169.314,51.632,159.906
C01334=1016.736,271.497,-136.916,169.309,51.638,159.906
C01335=1016.729,271.249,-136.887,169.304,51.644,159.907
C01336=1016.724,271.001,-136.858,169.298,51.650,159.907
C01337=1016.718,270.753,-136.829,169.293,51.657,159.908
C01338=1016.713,270.505,-136.799,169.288,51.663,159.908
C01339=1016.707,270.257,-136.770,169.283,51.669,159.908
C01340=1016.700,270.009,-136.741,169.278,51.674,159.909
C01341=1016.695,269.760,-136.712,169.274,51.681,159.909
C01342=1016.689,269.511,-136.683,169.268,51.687,159.910
C01343=1016.683,269.263,-136.654,169.263,51.693,159.910
C01344=1016.678,269.015,-136.625,169.258,51.699,159.910
C01345=1016.671,268.767,-136.596,169.253,51.705,159.911
C01346=1016.665,268.519,-136.567,169.248,51.711,159.911
C01347=1016.659,268.270,-136.539,169.243,51.718,159.912
C01348=1016.654,268.022,-136.509,169.238,51.724,159.912
C01349=1016.648,267.775,-136.480,169.233,51.730,159.913
C01350=1016.642,267.526,-136.452,169.228,51.737,159.913
C01351=1016.636,267.278,-136.423,169.222,51.743,159.913
C01352=1016.630,267.029,-136.393,169.218,51.749,159.914
C01353=1016.624,266.781,-136.365,169.213,51.755,159.914
C01354=1016.619,266.533,-136.336,169.208,51.762,159.915
C01355=1016.613,266.285,-136.307,169.202,51.768,159.915
C01356=1016.607,266.036,-136.279,169.198,51.775,159.916
C01357=1016.601,265.788,-136.249,169.193,51.780,159.916
C01358=1016.596,265.540,-136.221,169.188,51.787,159.917
C01359=1016.590,265.292,-136.192,169.182,51.793,159.917
C01360=1016.583,265.043,-136.163,169.178,51.800,159.918
C01361=1016.577,264.795,-136.135,169.173,51.806,159.918
C01362=1016.572,264.547,-136.106,169.168,51.812,159.919
C01363=1016.566,264.313,-136.079,169.164,51.819,159.919
C01364=1016.561,264.079,-136.052,169.159,51.825,159.920
C01365=1016.556,263.845,-136.026,169.154,51.831,159.920
C01366=1016.550,263.611,-135.999,169.149,51.837,159.921
C01367=1016.544,263.377,-135.972,169.144,51.843,159.921
C01368=1016.538,263.142,-135.945,169.140,51.849,159.922
C01369=1016.534,262.909,-135.918,169.136,51.855,159.922
C01370=1016.528,262.674,-135.891,169.131,51.861,159.923
C01371=1016.522,262.426,-135.863,169.126,51.868,159.923
C01372=1016.516,262.178,-135.834,169.121,51.875,159.924
C01373=1016.511,261.929,-135.806,169.116,51.881,159.924
C01374=1016.505,261.681,-135.778,169.112,51.887,159.925
C01375=1016.499,261.433,-135.749,169.106,51.894,159.925
C01376=1016.493,261.185,-135.721,169.101,51.901,159.926
C01377=1016.487,260.936,-135.692,169.097,51.907,159.926
C01378=1016.481,260.688,-135.664,169.091,51.914,159.927
C01379=1016.475,260.440,-135.635,169.087,51.921,159.928
C01380=1016.470,260.192,-135.607,169.082,51.927,159.928
C01381=1016.464,259.943,-135.579,169.076,51.933,159.928
C01382=1016.460,259.694,-135.551,169.072,51.940,159.929
C01383=1016.453,259.447,-135.522,169.067,51.947,159.930
C01384=1016.447,259.199,-135.494,169.062,51.954,159.930
C01385=1016.441,258.950,-135.466,169.057,51.960,159.931
C01386=1016.435,258.702,-135.438,169.053,51.967,159.932
C01387=1016.429,258.454,-135.411,169.048,51.974,159.932
C01388=1016.423,258.205,-135.382,169.043,51.981,159.933
C01389=1016.417,257.957,-135.354,169.038,51.988,159.933
C01390=1016.411,257.708,-135.327,169.033,51.994,159.934
C01391=1016.406,257.460,-135.299,169.028,52.001,159.934
C01392=1016.400,257.211,-135.271,169.023,52.008,159.935
C01393=1016.394,256.963,-135.244,169.019,52.015,159.936
C01394=1016.388,256.714,-135.215,169.014,52.022,159.936
C01395=1016.381,256.467,-135.188,169.009,52.029,159.937
C01396=1016.376,256.218,-135.160,169.004,52.036,159.937
C01397=1016.370,255.970,-135.132,168.999,52.043,159.938
C01398=1016.364,255.721,-135.105,168.994,52.050,159.939
C01399=1016.358,255.473,-135.077,168.989,52.057,159.939
C01400=1016.353,255.224,-135.048,168.985,52.063,159.940
C01401=1016.346,254.976,-135.021,168.980,52.071,159.940
C01402=1016.341,254.728,-134.993,168.975,52.078,159.941
C01403=1016.335,254.479,-134.966,168.970,52.084,159.942
C01404=1016.329,254.230,-134.938,168.966,52.092,159.942
C01405=1016.323,253.982,-134.910,168.960,52.099,159.943
C01406=1016.317,253.735,-134.883,168.956,52.105,159.943
C01407=1016.312,253.485,-134.855,168.951,52.113,159.944
C01408=1016.306,253.237,-134.827,168.946,52.120,159.945
C01409=1016.300,252.989,-134.799,168.941,52.127,159.945
C01410=1016.295,252.740,-134.772,168.937,52.134,159.946
C01411=1016.289,252.492,-134.745,168.932,52.141,159.947
C01412=1016.283,252.244,-134.716,168.927,52.148,159.947
C01413=1016.278,251.995,-134.689,168.923,52.155,159.948
C01414=1016.271,251.747,-134.661,168.917,52.162,159.949
C01415=1016.266,251.498,-134.634,168.913,52.169,159.949
C01416=1016.260,251.250,-134.607,168.907,52.176,159.950
C01417=1016.254,251.001,-134.578,168.903,52.183,159.951
C01418=1016.249,250.753,-134.551,168.898,52.190,159.951
C01419=1016.243,250.505,-134.524,168.894,52.198,159.952
C01420=1016.237,250.256,-134.496,168.889,52.205,159.953
C01421=1016.232,250.008,-134.468,168.884,52.212,159.953
C01422=1016.226,249.759,-134.442,168.879,52.220,159.954
C01423=1016.221,249.524,-134.415,168.875,52.226,159.954
C01424=1016.216,249.289,-134.389,168.870,52.233,159.955
C01425=1016.210,249.055,-134.363,168.866,52.240,159.956
C01426=1016.204,248.820,-134.337,168.861,52.246,159.956
C01427=1016.200,248.584,-134.311,168.857,52.253,159.957
C01428=1016.194,248.349,-134.286,168.853,52.260,159.958
C01429=1016.188,248.114,-134.259,168.848,52.267,159.958
C01430=1016.183,247.880,-134.233,168.844,52.274,159.959
C01431=1016.177,247.631,-134.206,168.839,52.281,159.960
C01432=1016.172,247.383,-134.178,168.835,52.288,159.960
C01433=1016.167,247.134,-134.151,168.830,52.296,159.961
C01434=1016.161,246.885,-134.124,168.825,52.303,159.962
C01435=1016.155,246.637,-134.096,168.820,52.310,159.962
C01436=1016.150,246.389,-134.069,168.816,52.318,159.963
C01437=1016.145,246.140,-134.042,168.811,52.325,159.964
C01438=1016.139,245.892,-134.014,168.807,52.332,159.965
C01439=1016.133,245.643,-133.987,168.802,52.340,159.965
C01440=1016.128,245.394,-133.960,168.798,52.347,159.966
C01441=1016.122,245.147,-133.933,168.792,52.354,159.967
C01442=1016.117,244.898,-133.905,168.788,52.361,159.967
C01443=1016.112,244.649,-133.878,168.783,52.369,159.968
C01444=1016.106,244.402,-133.851,168.779,52.376,159.969
C01445=1016.101,244.153,-133.823,168.774,52.384,159.970
C01446=1016.094,243.904,-133.796,168.768,52.391,159.970
C01447=1016.089,243.655,-133.769,168.764,52.399,159.971
C01448=1016.084,243.407,-133.741,168.759,52.406,159.972
C01449=1016.078,243.159,-133.715,168.755,52.414,159.972
C01450=1016.073,242.910,-133.687,168.750,52.421,159.973
C01451=1016.067,242.662,-133.661,168.746,52.429,159.974
C01452=1016.061,242.413,-133.634,168.741,52.436,159.975
C01453=1016.056,242.165,-133.607,168.736,52.444,159.975
C01454=1016.050,241.917,-133.579,168.732,52.451,159.976
C01455=1016.045,241.669,-133.553,168.727,52.459,159.977
C01456=1016.039,241.420,-133.526,168.723,52.466,159.978
C01457=1016.034,241.172,-133.499,168.718,52.474,159.978
C01458=1016.028,240.923,-133.472,168.713,52.482,159.979
C01459=1016.022,240.675,-133.446,168.709,52.489,159.980
C01460=1016.017,240.426,-133.418,168.704,52.497,159.981
C01461=1016.012,240.177,-133.392,168.699,52.505,159.981
C01462=1016.006,239.929,-133.366,168.696,52.513,159.982
C01463=1016.001,239.680,-133.339,168.691,52.521,159.983
C01464=1015.995,239.432,-133.312,168.685,52.528,159.984
C01465=1015.989,239.183,-133.285,168.681,52.536,159.985
C01466=1015.984,238.934,-133.258,168.676,52.543,159.985
C01467=1015.979,238.687,-133.231,168.672,52.552,159.986
C01468=1015.973,238.438,-133.205,168.668,52.559,159.987
C01469=1015.967,238.190,-133.178,168.663,52.567,159.988
C01470=1015.961,237.941,-133.152,168.658,52.575,159.989
C01471=1015.956,237.692,-133.125,168.653,52.583,159.989
C01472=1015.950,237.444,-133.099,168.649,52.590,159.990
C01473=1015.944,237.195,-133.073,168.645,52.599,159.991
C01474=1015.939,236.947,-133.046,168.640,52.607,159.992
C01475=1015.933,236.698,-133.020,168.635,52.614,159.992
C01476=1015.927,236.450,-132.993,168.631,52.622,159.994
C01477=1015.922,236.201,-132.967,168.626,52.630,159.994
C01478=1015.916,235.953,-132.940,168.622,52.639,159.995
C01479=1015.910,235.704,-132.914,168.617,52.646,159.996
C01480=1015.905,235.455,-132.888,168.613,52.654,159.997
C01481=1015.899,235.207,-132.861,168.608,52.662,159.998
C01482=1015.893,234.958,-132.835,168.604,52.671,159.999
C01483=1015.888,234.720,-132.810,168.599,52.678,159.999
C01484=1015.883,234.481,-132.785,168.595,52.686,160.000
C01485=1015.877,234.244,-132.759,168.590,52.693,160.001
C01486=1015.872,234.005,-132.734,168.586,52.702,160.002
C01487=1015.866,233.767,-132.709,168.581,52.709,160.003
C01488=1015.862,233.528,-132.684,168.577,52.717,160.003
C01489=1015.856,233.290,-132.659,168.573,52.725,160.004
C01490=1015.851,233.052,-132.634,168.569,52.733,160.005
C01491=1015.845,232.804,-132.607,168.564,52.740,160.006
C01492=1015.840,232.555,-132.581,168.559,52.749,160.007
C01493=1015.834,232.306,-132.556,168.554,52.757,160.008
C01494=1015.828,232.057,-132.529,168.551,52.765,160.008
C01495=1015.823,231.809,-132.503,168.546,52.773,160.009
C01496=1015.818,231.561,-132.477,168.541,52.782,160.010
C01497=1015.812,231.312,-132.451,168.536,52.789,160.011
C01498=1015.806,231.063,-132.424,168.532,52.798,160.012
C01499=1015.801,230.813,-132.398,168.527,52.806,160.013
C01500=1015.795,230.564,-132.373,168.523,52.815,160.014
C01501=1015.790,230.314,-132.346,168.519,52.822,160.015
C01502=1015.784,230.065,-132.320,168.514,52.831,160.016
C01503=1015.779,229.816,-132.294,168.510,52.839,160.016
C01504=1015.773,229.567,-132.268,168.505,52.848,160.017
C01505=1015.768,229.319,-132.242,168.501,52.856,160.018
C01506=1015.762,229.071,-132.216,168.496,52.865,160.019
C01507=1015.757,228.822,-132.190,168.491,52.872,160.020
C01508=1015.751,228.573,-132.164,168.487,52.881,160.021
C01509=1015.746,228.325,-132.138,168.482,52.889,160.022
C01510=1015.741,228.076,-132.112,168.478,52.898,160.023
C01511=1015.734,227.827,-132.087,168.473,52.906,160.024
C01512=1015.729,227.578,-132.061,168.469,52.915,160.025
C01513=1015.724,227.330,-132.035,168.464,52.923,160.026
C01514=1015.718,227.082,-132.009,168.461,52.931,160.027
C01515=1015.713,226.833,-131.983,168.456,52.940,160.027
C01516=1015.708,226.585,-131.957,168.452,52.948,160.028
C01517=1015.702,226.336,-131.932,168.447,52.957,160.029
C01518=1015.696,226.087,-131.906,168.443,52.965,160.030
C01519=1015.691,225.839,-131.881,168.438,52.974,160.031
C01520=1015.685,225.590,-131.855,168.434,52.982,160.032
C01521=1015.680,225.341,-131.829,168.429,52.992,160.033
C01522=1015.673,225.092,-131.804,168.424,53.000,160.034
C01523=1015.669,224.844,-131.778,168.420,53.009,160.035
C01524=1015.662,224.595,-131.753,168.415,53.017,160.036
C01525=1015.657,224.346,-131.727,168.411,53.026,160.037
C01526=1015.651,224.098,-131.702,168.407,53.035,160.038
C01527=1015.646,223.849,-131.677,168.402,53.044,160.039
C01528=1015.641,223.601,-131.652,168.398,53.052,160.040
C01529=1015.635,223.352,-131.626,168.393,53.061,160.041
C01530=1015.630,223.103,-131.600,168.389,53.070,160.042
C01531=1015.624,222.855,-131.575,168.385,53.078,160.043
C01532=1015.619,222.606,-131.549,168.380,53.087,160.044
C01533=1015.612,222.357,-131.524,168.375,53.097,160.045
C01534=1015.608,222.108,-131.499,168.371,53.105,160.046
C01535=1015.602,221.860,-131.473,168.366,53.114,160.047
C01536=1015.597,221.611,-131.448,168.362,53.123,160.048
C01537=1015.590,221.363,-131.423,168.358,53.131,160.049
C01538=1015.586,221.114,-131.397,168.353,53.140,160.050
C01539=1015.580,220.865,-131.372,168.349,53.149,160.051
C01540=1015.574,220.616,-131.346,168.345,53.158,160.052
C01541=1015.569,220.368,-131.321,168.341,53.167,160.053
C01542=1015.563,220.119,-131.296,168.335,53.176,160.054
C01543=1015.558,219.877,-131.271,168.331,53.184,160.055
C01544=1015.553,219.636,-131.247,168.327,53.192,160.056
C01545=1015.547,219.393,-131.222,168.324,53.202,160.057
C01546=1015.543,219.151,-131.197,168.319,53.210,160.058
C01547=1015.537,218.909,-131.172,168.315,53.219,160.059
C01548=1015.532,218.667,-131.148,168.310,53.227,160.060
C01549=1015.527,218.426,-131.124,168.306,53.237,160.061
C01550=1015.521,218.184,-131.099,168.302,53.245,160.062
C01551=1015.517,217.935,-131.074,168.297,53.254,160.063
C01552=1015.510,217.686,-131.049,168.292,53.263,160.064
C01553=1015.505,217.438,-131.024,168.288,53.273,160.065
C01554=1015.499,217.189,-130.999,168.284,53.281,160.066
C01555=1015.494,216.940,-130.974,168.280,53.290,160.067
C01556=1015.489,216.692,-130.949,168.275,53.300,160.068
C01557=1015.482,216.443,-130.924,168.271,53.309,160.069
C01558=1015.477,216.195,-130.900,168.266,53.318,160.070
C01559=1015.471,215.945,-130.875,168.261,53.327,160.071
C01560=1015.466,215.697,-130.850,168.257,53.337,160.072
C01561=1015.460,215.448,-130.825,168.254,53.346,160.074
C01562=1015.455,215.200,-130.800,168.250,53.355,160.075
C01563=1015.449,214.951,-130.775,168.244,53.364,160.076
C01564=1015.444,214.702,-130.750,168.240,53.373,160.077
C01565=1015.439,214.454,-130.725,168.236,53.383,160.078
C01566=1015.433,214.204,-130.701,168.231,53.392,160.079
C01567=1015.427,213.956,-130.676,168.227,53.402,160.080
C01568=1015.422,213.707,-130.651,168.223,53.411,160.081
C01569=1015.417,213.458,-130.626,168.218,53.421,160.082
C01570=1015.411,213.210,-130.601,168.214,53.429,160.083
C01571=1015.405,212.961,-130.577,168.209,53.439,160.084
C01572=1015.401,212.712,-130.552,168.205,53.448,160.085
C01573=1015.395,212.463,-130.528,168.201,53.457,160.087
C01574=1015.389,212.215,-130.502,168.196,53.467,160.088
C01575=1015.384,211.966,-130.478,168.192,53.476,160.089
C01576=1015.379,211.717,-130.453,168.188,53.486,160.090
C01577=1015.373,211.469,-130.428,168.183,53.495,160.091
C01578=1015.368,211.220,-130.404,168.179,53.505,160.092
C01579=1015.363,210.971,-130.379,168.174,53.514,160.093
C01580=1015.357,210.722,-130.355,168.170,53.523,160.094
C01581=1015.352,210.473,-130.330,168.167,53.533,160.096
C01582=1015.347,210.225,-130.305,168.162,53.542,160.097
C01583=1015.341,209.976,-130.280,168.158,53.552,160.098
C01584=1015.335,209.727,-130.256,168.153,53.561,160.099
C01585=1015.331,209.479,-130.231,168.149,53.571,160.100
C01586=1015.325,209.230,-130.207,168.144,53.581,160.101
C01587=1015.320,208.981,-130.182,168.140,53.590,160.102
C01588=1015.314,208.733,-130.157,168.135,53.600,160.104
C01589=1015.309,208.484,-130.133,168.132,53.609,160.105
C01590=1015.303,208.236,-130.109,168.127,53.620,160.106
C01591=1015.297,207.986,-130.084,168.123,53.629,160.107
C01592=1015.292,207.738,-130.060,168.118,53.639,160.108
C01593=1015.287,207.489,-130.036,168.114,53.648,160.109
C01594=1015.282,207.240,-130.011,168.110,53.659,160.111
C01595=1015.276,206.991,-129.987,168.106,53.668,160.112
C01596=1015.270,206.743,-129.963,168.101,53.678,160.113
C01597=1015.265,206.494,-129.938,168.098,53.688,160.114
C01598=1015.260,206.245,-129.914,168.093,53.697,160.115
C01599=1015.255,205.996,-129.891,168.088,53.707,160.116
C01600=1015.249,205.747,-129.866,168.084,53.717,160.118
C01601=1015.244,205.498,-129.842,168.080,53.727,160.119
C01602=1015.238,205.250,-129.817,168.076,53.737,160.120
C01603=1015.233,205.017,-129.795,168.072,53.746,160.121
C01604=1015.227,204.783,-129.772,168.068,53.755,160.122
C01605=1015.223,204.550,-129.750,168.063,53.765,160.123
C01606=1015.218,204.317,-129.727,168.059,53.774,160.125
C01607=1015.213,204.084,-129.705,168.055,53.783,160.126
C01608=1015.207,203.851,-129.682,168.051,53.793,160.127
C01609=1015.202,203.618,-129.660,168.047,53.802,160.128
C01610=1015.197,203.385,-129.638,168.044,53.811,160.129
C01611=1015.178,202.296,-129.540,167.527,53.748,160.004
C01612=1015.174,202.048,-129.517,167.522,53.758,160.005
C01613=1015.169,201.799,-129.495,167.518,53.770,160.007
C01614=1015.165,201.550,-129.472,167.513,53.781,160.008
C01615=1015.161,201.301,-129.450,167.508,53.792,160.009
C01616=1015.156,201.052,-129.428,167.503,53.803,160.010
C01617=1015.152,200.803,-129.406,167.499,53.814,160.012
C01618=1015.148,200.554,-129.383,167.493,53.825,160.013
C01619=1015.143,200.305,-129.361,167.489,53.836,160.014
C01620=1015.139,200.056,-129.339,167.484,53.848,160.016
C01621=1015.135,199.807,-129.316,167.480,53.858,160.017
C01622=1015.130,199.558,-129.294,167.475,53.870,160.018
C01623=1015.126,199.309,-129.272,167.470,53.880,160.019
C01624=1015.122,199.060,-129.250,167.466,53.892,160.021
C01625=1015.117,198.811,-129.228,167.461,53.903,160.022
C01626=1015.112,198.562,-129.206,167.456,53.915,160.023
C01627=1015.108,198.313,-129.183,167.452,53.925,160.025
C01628=1015.103,198.064,-129.161,167.447,53.937,160.026
C01629=1015.098,197.815,-129.140,167.443,53.948,160.027
C01630=1015.094,197.565,-129.118,167.438,53.960,160.029
C01631=1015.090,197.317,-129.096,167.434,53.971,160.030
C01632=1015.085,197.068,-129.074,167.428,53.982,160.031
C01633=1015.080,196.819,-129.052,167.423,53.993,160.032
C01634=1015.076,196.569,-129.031,167.419,54.005,160.034
C01635=1015.071,196.320,-129.009,167.414,54.016,160.035
C01636=1015.067,196.072,-128.987,167.410,54.027,160.037
C01637=1015.063,195.823,-128.965,167.405,54.039,160.038
C01638=1015.059,195.574,-128.944,167.401,54.050,160.039
C01639=1015.054,195.325,-128.922,167.396,54.061,160.040
C01640=1015.049,195.076,-128.901,167.392,54.072,160.042
C01641=1015.045,194.826,-128.878,167.387,54.084,160.043
C01642=1015.040,194.578,-128.856,167.383,54.095,160.045
C01643=1015.036,194.328,-128.835,167.377,54.106,160.046
C01644=1015.032,194.080,-128.813,167.374,54.117,160.047
C01645=1015.027,193.831,-128.791,167.369,54.129,160.048
C01646=1015.023,193.582,-128.770,167.365,54.140,160.050
C01647=1015.018,193.333,-128.748,167.361,54.152,160.051
C01648=1015.014,193.084,-128.726,167.355,54.163,160.052
C01649=1015.009,192.834,-128.705,167.351,54.174,160.054
C01650=1015.005,192.586,-128.683,167.346,54.185,160.055
C01651=1015.001,192.336,-128.661,167.342,54.197,160.057
C01652=1014.997,192.087,-128.639,167.337,54.208,160.058
C01653=1014.992,191.838,-128.618,167.333,54.219,160.059
C01654=1014.988,191.590,-128.597,167.329,54.230,160.061
C01655=1014.984,191.340,-128.575,167.324,54.242,160.062
C01656=1014.979,191.091,-128.553,167.320,54.253,160.063
C01657=1014.975,190.842,-128.532,167.315,54.264,160.064
C01658=1014.971,190.594,-128.511,167.311,54.275,160.066
C01659=1014.967,190.344,-128.489,167.307,54.287,160.067
C01660=1014.962,190.095,-128.467,167.302,54.298,160.069
C01661=1014.957,189.846,-128.446,167.298,54.309,160.070
C01662=1014.954,189.597,-128.424,167.293,54.321,160.071
C01663=1014.949,189.348,-128.403,167.289,54.332,160.073
C01664=1014.945,189.099,-128.381,167.285,54.343,160.074
C01665=1014.940,188.850,-128.359,167.280,54.355,160.075
C01666=1014.937,188.601,-128.337,167.276,54.365,160.077
C01667=1014.932,188.352,-128.316,167.272,54.377,160.078
C01668=1014.928,188.102,-128.295,167.267,54.388,160.079
C01669=1014.923,187.854,-128.274,167.263,54.400,160.081
C01670=1014.920,187.605,-128.252,167.259,54.410,160.082
C01671=1014.915,187.356,-128.230,167.254,54.422,160.083
C01672=1014.910,187.076,-128.206,167.249,54.434,160.085
C01673=1014.906,186.797,-128.182,167.245,54.447,160.086
C01674=1014.901,186.517,-128.159,167.239,54.460,160.088
C01675=1014.896,186.238,-128.134,167.235,54.472,160.089
C01676=1014.892,185.988,-128.112,167.230,54.484,160.091
C01677=1014.888,185.739,-128.092,167.226,54.495,160.092
C01678=1014.883,185.491,-128.070,167.222,54.506,160.094
C01679=1014.879,185.241,-128.049,167.218,54.517,160.095
C01680=1014.876,184.992,-128.027,167.213,54.529,160.096
C01681=1014.871,184.743,-128.006,167.209,54.540,160.098
C01682=1014.867,184.495,-127.985,167.205,54.551,160.099
C01683=1014.862,184.245,-127.963,167.201,54.562,160.100
C01684=1014.859,183.996,-127.942,167.196,54.574,160.102
C01685=1014.855,183.747,-127.921,167.193,54.585,160.103
C01686=1014.850,183.498,-127.899,167.188,54.596,160.104
C01687=1014.846,183.249,-127.878,167.184,54.607,160.106
C01688=1014.842,182.999,-127.857,167.181,54.618,160.107
C01689=1014.838,182.751,-127.836,167.175,54.629,160.108
C01690=1014.834,182.502,-127.814,167.171,54.641,160.110
C01691=1014.830,182.253,-127.793,167.168,54.652,160.111
C01692=1014.826,182.003,-127.771,167.164,54.663,160.113
C01693=1014.821,181.754,-127.750,167.159,54.674,160.114
C01694=1014.817,181.505,-127.729,167.155,54.686,160.115
C01695=1014.813,181.256,-127.708,167.151,54.697,160.117
C01696=1014.809,181.007,-127.688,167.147,54.709,160.118
C01697=1014.804,180.757,-127.668,167.142,54.720,160.119
C01698=1014.800,180.509,-127.647,167.138,54.732,160.121
C01699=1014.795,180.259,-127.626,167.135,54.743,160.122
C01700=1014.791,180.011,-127.606,167.130,54.755,160.124
C01701=1014.786,179.761,-127.584,167.126,54.766,160.125
C01702=1014.782,179.512,-127.565,167.121,54.778,160.126
C01703=1014.778,179.263,-127.544,167.117,54.789,160.128
C01704=1014.773,179.014,-127.524,167.114,54.801,160.129
C01705=1014.768,178.765,-127.502,167.109,54.813,160.131
C01706=1014.765,178.516,-127.482,167.105,54.824,160.132
C01707=1014.759,178.266,-127.462,167.101,54.835,160.134
C01708=1014.756,178.018,-127.441,167.097,54.847,160.135
C01709=1014.751,177.768,-127.421,167.093,54.859,160.136
C01710=1014.747,177.519,-127.400,167.089,54.870,160.138
C01711=1014.742,177.270,-127.379,167.085,54.881,160.139
C01712=1014.738,177.021,-127.359,167.081,54.893,160.141
C01713=1014.733,176.771,-127.339,167.077,54.905,160.142
C01714=1014.729,176.523,-127.318,167.073,54.916,160.144
C01715=1014.724,176.274,-127.297,167.068,54.928,160.145
C01716=1014.721,176.024,-127.277,167.065,54.939,160.146
C01717=1014.716,175.776,-127.257,167.061,54.951,160.148
C01718=1014.712,175.526,-127.237,167.057,54.962,160.149
C01719=1014.707,175.277,-127.216,167.052,54.974,160.151
C01720=1014.703,175.028,-127.195,167.049,54.985,160.152
C01721=1014.699,174.778,-127.175,167.045,54.997,160.154
C01722=1014.694,174.530,-127.155,167.041,55.008,160.155
C01723=1014.690,174.280,-127.135,167.036,55.020,160.156
C01724=1014.685,174.032,-127.114,167.033,55.031,160.158
C01725=1014.681,173.783,-127.094,167.029,55.043,160.159
C01726=1014.677,173.533,-127.073,167.025,55.054,160.161
C01727=1014.673,173.284,-127.053,167.020,55.065,160.162
C01728=1014.668,173.034,-127.033,167.016,55.077,160.163
C01729=1014.664,172.786,-127.012,167.013,55.088,160.165
C01730=1014.660,172.537,-126.992,167.009,55.100,160.166
C01731=1014.655,172.287,-126.972,167.005,55.111,160.168
C01732=1014.651,172.038,-126.952,167.002,55.123,160.169
C01733=1014.647,171.789,-126.931,166.997,55.135,160.171
C01734=1014.642,171.540,-126.911,166.993,55.146,160.172
C01735=1014.638,171.291,-126.890,166.990,55.157,160.174
C01736=1014.634,171.011,-126.868,166.985,55.170,160.175
C01737=1014.630,170.731,-126.845,166.981,55.183,160.177
C01738=1014.624,170.451,-126.822,166.976,55.196,160.178
C01739=1014.619,170.172,-126.799,166.972,55.209,160.180
C01740=1014.616,169.923,-126.779,166.968,55.220,160.181
C01741=1014.610,169.674,-126.759,166.964,55.231,160.183
C01742=1014.607,169.424,-126.739,166.961,55.243,160.184
C01743=1014.603,169.175,-126.719,166.957,55.254,160.186
C01744=1014.598,168.927,-126.699,166.952,55.266,160.187
C01745=1014.594,168.677,-126.678,166.949,55.277,160.189
C01746=1014.590,168.428,-126.658,166.945,55.289,160.190
C01747=1014.586,168.179,-126.638,166.941,55.300,160.191
C01748=1014.582,167.929,-126.618,166.937,55.311,160.193
C01749=1014.577,167.680,-126.597,166.934,55.323,160.194
C01750=1014.574,167.431,-126.577,166.930,55.334,160.196
C01751=1014.569,167.182,-126.558,166.927,55.346,160.197
C01752=1014.565,166.933,-126.537,166.923,55.357,160.199
C01753=1014.561,166.684,-126.517,166.919,55.368,160.200
C01754=1014.556,166.435,-126.496,166.915,55.379,160.201
C01755=1014.553,166.185,-126.476,166.912,55.391,160.203
C01756=1014.548,165.936,-126.457,166.908,55.402,160.204
C01757=1014.545,165.687,-126.437,166.904,55.414,160.206
C01758=1014.540,165.439,-126.416,166.900,55.425,160.207
C01759=1014.537,165.189,-126.396,166.897,55.436,160.209
C01760=1014.532,164.939,-126.377,166.893,55.448,160.210
C01761=1014.528,164.691,-126.356,166.889,55.459,160.212
C01762=1014.524,164.441,-126.336,166.886,55.471,160.213
C01763=1014.520,164.192,-126.316,166.882,55.482,160.214
C01764=1014.516,163.943,-126.296,166.878,55.493,160.216
C01765=1014.511,163.695,-126.276,166.875,55.505,160.217
C01766=1014.508,163.445,-126.256,166.871,55.516,160.219
C01767=1014.504,163.195,-126.236,166.867,55.527,160.220
C01768=1014.499,162.946,-126.216,166.863,55.539,160.222
C01769=1014.495,162.697,-126.195,166.860,55.550,160.223
C01770=1014.491,162.448,-126.176,166.856,55.562,160.225
C01771=1014.487,162.199,-126.156,166.852,55.573,160.226
C01772=1014.483,161.950,-126.136,166.849,55.584,160.227
C01773=1014.479,161.701,-126.116,166.845,55.596,160.229
C01774=1014.476,161.452,-126.095,166.842,55.607,160.230
C01775=1014.471,161.203,-126.076,166.837,55.618,160.231
C01776=1014.468,160.953,-126.056,166.835,55.629,160.233
C01777=1014.463,160.704,-126.036,166.831,55.641,160.235
